fbTrendLogger(
    VI_System_Time_MS := GVL_TIME_SERVICE.G_Now_MS,
    VI_Config := L_TrendConfig,
    VI_Current_Value := GVL_STATE.G_Room_Temps[1],
    VO_Data => L_TrendData
);

fbTrendAdapter(
    VI_Data := L_TrendData,
    VO_Average => L_Average,
    VO_Min => L_Min,
    VO_Max => L_Max,
    VO_Trend_Up => L_Trend_Up,
    VO_Trend_Down => L_Trend_Down
);
          
END_PROGRAM

PROGRAM PRG_Peer_Session_Publication

            // ======================================================
// PEER SESSION PUBLICATION
// ======================================================
// Canonical local PLC session export.
//
// Purpose:
// publish normalized runtime/session authority state into
// explicit peer-session transport contract surface.
//
// This layer does NOT:
// - perform network replication
// - perform distributed reconciliation
// - consume remote peer state
//
// Future transport/replication layers may replicate these
// fields to partner PLCs or external HA channels.
// ======================================================

GVL_PEER_SESSION.Remote_Session_Valid :=
    GVL_RUNTIME_EPOCH.Runtime_Runtime_Barrier_OK
    AND GVL_RUNTIME_EPOCH.Runtime_IO_Publication_Allowed;

GVL_PEER_SESSION.Remote_Last_Refresh_MS :=
    GVL_STATUS.G_System_Time_MS;

GVL_PEER_SESSION.Remote_Runtime_Epoch :=
    GVL_RUNTIME_EPOCH.Runtime_Epoch;

GVL_PEER_SESSION.Remote_Snapshot_Epoch :=
    GVL_RUNTIME_SNAPSHOT.Snapshot_Epoch;

GVL_PEER_SESSION.Remote_Boot_Generation :=
    GVL_TIME_MONOTONIC.Boot_Generation_ID;

GVL_PEER_SESSION.Remote_Fencing_Token :=
    GVL_PLC_FENCING.PLC_Fencing_Token;

GVL_PEER_SESSION.Remote_Publication_Allowed :=
    GVL_OUTPUT_EPOCH.Output_Publication_Valid
    AND NOT GVL_OUTPUT_EPOCH.Output_Forced_Safe_Decay;

GVL_PEER_SESSION.Remote_Runtime_Healthy :=
    GVL_RUNTIME_EPOCH.Runtime_Runtime_Barrier_OK;

// >>> BULK_SYNC_ANCHOR: PRG_Peer_Session_Publication <<<
          
END_PROGRAM

PROGRAM PRG_PLC_Arbitration

            // Update heartbeat
IF GVL_STATUS.G_Remote_PLC_Pulse THEN
    GVL_STATUS.G_Remote_PLC_Last_Seen_MS := GVL_TIME_SERVICE.G_Now_MS;
END_IF;

// Alive check (3s)
GVL_STATUS.G_Remote_PLC_Alive :=
    (GVL_TIME_SERVICE.G_Now_MS - GVL_STATUS.G_Remote_PLC_Last_Seen_MS) < 3000;

// Deterministic arbitration.
// If remote is not alive, local PLC owns runtime.
// If remote is alive, the lowest PLC ID wins; equality keeps local active
// because G_Active_PLC_ID defaults to the configured local owner ID.
IF NOT GVL_STATUS.G_Remote_PLC_Alive THEN
    GVL_STATUS.G_Is_Active_PLC := TRUE;
    GVL_STATUS.G_Active_PLC_ID := GVL_STATUS.G_Local_PLC_ID;
ELSE
    IF GVL_STATUS.G_Local_PLC_ID <= GVL_STATUS.G_Active_PLC_ID THEN
        GVL_STATUS.G_Is_Active_PLC := TRUE;
        GVL_STATUS.G_Active_PLC_ID := GVL_STATUS.G_Local_PLC_ID;
    ELSE
        GVL_STATUS.G_Is_Active_PLC := FALSE;
    END_IF;
END_IF;

GVL_STATUS.G_Other_PLC_Is_Active :=
    GVL_STATUS.G_Remote_PLC_Alive AND NOT GVL_STATUS.G_Is_Active_PLC;

// >>> BULK_SYNC_ANCHOR: PRG_PLC_Arbitration <<<
          
END_PROGRAM

PROGRAM PRG_Physical_Snapshot_Governor
  VAR
    L_Now_MS : UDINT;
    L_Snapshot_Valid : BOOL := TRUE;
    L_Error_Code : UDINT := 0;
    L_Error_Text : STRING(160) := '';
  END_VAR

            L_Now_MS := GVL_STATUS.G_System_Time_MS;
L_Snapshot_Valid := TRUE;
L_Error_Code := 0;
L_Error_Text := '';

GVL_PHYSICAL_SNAPSHOT.Physical_Snapshot_Valid := FALSE;
GVL_PHYSICAL_SNAPSHOT.Physical_Snapshot_Frozen := FALSE;
GVL_PHYSICAL_SNAPSHOT.Physical_Snapshot_Publication_Allowed := FALSE;
GVL_PHYSICAL_SNAPSHOT.Physical_Snapshot_Isolation_Valid := FALSE;
GVL_PHYSICAL_SNAPSHOT.Physical_Snapshot_Copy_Valid := FALSE;
GVL_PHYSICAL_SNAPSHOT.Physical_Snapshot_Freshness_Valid := FALSE;
GVL_PHYSICAL_SNAPSHOT.Physical_Snapshot_Consensus_Coherent := FALSE;
GVL_PHYSICAL_SNAPSHOT.Physical_Snapshot_Causality_Coherent := FALSE;

GVL_PHYSICAL_SNAPSHOT.Physical_Snapshot_Runtime_Epoch := ULINT_TO_UDINT(GVL_RUNTIME_EPOCH.Runtime_Epoch);
GVL_PHYSICAL_SNAPSHOT.Physical_Snapshot_Output_Epoch := ULINT_TO_UDINT(GVL_OUTPUT_EPOCH.Output_Publication_Epoch);

IF NOT GVL_RUNTIME_EPOCH.Runtime_Runtime_Barrier_OK THEN
    L_Snapshot_Valid := FALSE;
    L_Error_Code := 23000;
    L_Error_Text := 'Physical snapshot runtime barrier invalid';
END_IF;

IF L_Snapshot_Valid AND NOT GVL_OUTPUT_EPOCH.Output_Publication_Valid THEN
    L_Snapshot_Valid := FALSE;
    L_Error_Code := 23001;
    L_Error_Text := 'Physical snapshot output publication invalid';
END_IF;

IF L_Snapshot_Valid AND GVL_PHYSICAL_SNAPSHOT.Physical_Snapshot_Mutation_Detected THEN
    L_Snapshot_Valid := FALSE;
    L_Error_Code := 23002;
    L_Error_Text := 'Physical snapshot mutation detected';
END_IF;

IF L_Snapshot_Valid AND GVL_PHYSICAL_SNAPSHOT.Physical_Snapshot_Replay_Suspected THEN
    L_Snapshot_Valid := FALSE;
    L_Error_Code := 23003;
    L_Error_Text := 'Physical snapshot replay suspected';
END_IF;

IF L_Snapshot_Valid AND GVL_PHYSICAL_SNAPSHOT.Physical_Snapshot_Lease_Expired THEN
    L_Snapshot_Valid := FALSE;
    L_Error_Code := 23004;
    L_Error_Text := 'Physical snapshot lease expired';
END_IF;

IF L_Snapshot_Valid THEN
    GVL_PHYSICAL_SNAPSHOT.Physical_Snapshot_Valid := TRUE;
    GVL_PHYSICAL_SNAPSHOT.Physical_Snapshot_Frozen := TRUE;
    GVL_PHYSICAL_SNAPSHOT.Physical_Snapshot_Publication_Allowed := TRUE;
    GVL_PHYSICAL_SNAPSHOT.Physical_Snapshot_Isolation_Valid := TRUE;
    GVL_PHYSICAL_SNAPSHOT.Physical_Snapshot_Copy_Valid := TRUE;
    GVL_PHYSICAL_SNAPSHOT.Physical_Snapshot_Freshness_Valid := TRUE;
    GVL_PHYSICAL_SNAPSHOT.Physical_Snapshot_Consensus_Coherent := TRUE;
    GVL_PHYSICAL_SNAPSHOT.Physical_Snapshot_Causality_Coherent := TRUE;
    GVL_PHYSICAL_SNAPSHOT.Physical_Snapshot_Epoch := GVL_PHYSICAL_SNAPSHOT.Physical_Snapshot_Epoch + 1;
    GVL_PHYSICAL_SNAPSHOT.Physical_Snapshot_Last_Update_MS := L_Now_MS;
    GVL_PHYSICAL_SNAPSHOT.Physical_Snapshot_Last_Error_Code := 0;
    GVL_PHYSICAL_SNAPSHOT.Physical_Snapshot_Last_Error_Text := '';
ELSE
    GVL_PHYSICAL_SNAPSHOT.Physical_Snapshot_Valid := FALSE;
    GVL_PHYSICAL_SNAPSHOT.Physical_Snapshot_Frozen := FALSE;
    GVL_PHYSICAL_SNAPSHOT.Physical_Snapshot_Publication_Allowed := FALSE;
    GVL_PHYSICAL_SNAPSHOT.Physical_Snapshot_Last_Error_Code := L_Error_Code;
    GVL_PHYSICAL_SNAPSHOT.Physical_Snapshot_Last_Error_Text := L_Error_Text;
    GVL_PHYSICAL_SNAPSHOT.Physical_Snapshot_Invalidation_Count := GVL_PHYSICAL_SNAPSHOT.Physical_Snapshot_Invalidation_Count + 1;
END_IF;
          
END_PROGRAM

PROGRAM PRG_Causality_Reversal_Prevention_Governor

            IF GVL_HISTORICAL_ORDERING_INTEGRITY_FABRIC.Historical_Ordering_Integrity_Granted
AND NOT GVL_CAUSALITY_REVERSAL_PREVENTION_FABRIC.Causality_Reversal_Detected
AND NOT GVL_CAUSALITY_REVERSAL_PREVENTION_FABRIC.Resurrection_After_Revocation_Detected
AND NOT GVL_CAUSALITY_REVERSAL_PREVENTION_FABRIC.Unsafe_Temporal_Replay_Detected THEN

    GVL_CAUSALITY_REVERSAL_PREVENTION_FABRIC.Causality_Reversal_Prevention_Valid := TRUE;
    GVL_CAUSALITY_REVERSAL_PREVENTION_FABRIC.Causality_Reversal_Prevention_Granted := TRUE;
    GVL_CAUSALITY_REVERSAL_PREVENTION_FABRIC.Causality_Reversal_Prevented := TRUE;
    GVL_CAUSALITY_REVERSAL_PREVENTION_FABRIC.Authority_Ordering_Canonical := TRUE;
    GVL_CAUSALITY_REVERSAL_PREVENTION_FABRIC.Revocation_Resurrection_Boundary_Stable := TRUE;
END_IF;
          
END_PROGRAM

PROGRAM PRG_Epistemic_Integrity_Governor
  VAR
    L_Now_MS : UDINT;
    L_Epistemic_Valid : BOOL := TRUE;
    L_Error_Code : UDINT := 0;
    L_Error_Text : STRING(160) := '';
  END_VAR

            L_Now_MS := GVL_STATUS.G_System_Time_MS;
L_Epistemic_Valid := TRUE;
L_Error_Code := 0;
L_Error_Text := '';

// Fail-safe defaults.
GVL_EPISTEMIC_INTEGRITY_FABRIC.Epistemic_Integrity_Valid := FALSE;
GVL_EPISTEMIC_INTEGRITY_FABRIC.Epistemic_Integrity_Granted := FALSE;
GVL_EPISTEMIC_INTEGRITY_FABRIC.Epistemic_Integrity_Quarantine_Active := TRUE;

GVL_EPISTEMIC_INTEGRITY_FABRIC.Physical_Reality_Model_Coherent := FALSE;
GVL_EPISTEMIC_INTEGRITY_FABRIC.Sensor_Truth_Consensus_Valid := FALSE;
GVL_EPISTEMIC_INTEGRITY_FABRIC.Telemetry_Reality_Alignment_Stable := FALSE;
GVL_EPISTEMIC_INTEGRITY_FABRIC.Distributed_Reality_Model_Consistent := FALSE;
GVL_EPISTEMIC_INTEGRITY_FABRIC.Causal_Model_Physically_Valid := FALSE;

// Forensic evidence required.
IF NOT GVL_FORENSIC_EVIDENCE_FABRIC.Forensic_Evidence_Granted THEN
    L_Epistemic_Valid := FALSE;
    L_Error_Code := 44000;
    L_Error_Text := 'Forensic evidence authority not granted';
END_IF;

// Epistemic split-brain detectors.
IF GVL_EPISTEMIC_INTEGRITY_FABRIC.Physically_False_Consensus_Detected THEN
    L_Epistemic_Valid := FALSE;
    L_Error_Code := 44001;
    L_Error_Text := 'Physically false consensus detected';
END_IF;

IF GVL_EPISTEMIC_INTEGRITY_FABRIC.Telemetry_Corruption_Coherent_Detected THEN
    L_Epistemic_Valid := FALSE;
    L_Error_Code := 44002;
    L_Error_Text := 'Telemetry corruption coherence detected';
END_IF;

IF GVL_EPISTEMIC_INTEGRITY_FABRIC.Historical_Reality_Divergence_Detected THEN
    L_Epistemic_Valid := FALSE;
    L_Error_Code := 44003;
    L_Error_Text := 'Historical reality divergence detected';
END_IF;

IF GVL_EPISTEMIC_INTEGRITY_FABRIC.Sensor_Trust_Erosion_Detected THEN
    L_Epistemic_Valid := FALSE;
    L_Error_Code := 44004;
    L_Error_Text := 'Sensor trust erosion detected';
END_IF;

IF GVL_EPISTEMIC_INTEGRITY_FABRIC.Causal_Model_Poisoning_Detected THEN
    L_Epistemic_Valid := FALSE;
    L_Error_Code := 44005;
    L_Error_Text := 'Causal model poisoning detected';
END_IF;

IF GVL_EPISTEMIC_INTEGRITY_FABRIC.LongTerm_Epistemic_Drift_Detected THEN
    L_Epistemic_Valid := FALSE;
    L_Error_Code := 44006;
    L_Error_Text := 'Long-term epistemic drift detected';
END_IF;

// Physical reality anchoring validation.
IF L_Epistemic_Valid
AND NOT GVL_EPISTEMIC_INTEGRITY_FABRIC.Historical_Reality_Anchoring_Valid THEN
    L_Epistemic_Valid := FALSE;
    L_Error_Code := 44010;
    L_Error_Text := 'Historical reality anchoring invalid';
END_IF;

IF L_Epistemic_Valid
AND NOT GVL_EPISTEMIC_INTEGRITY_FABRIC.Physical_Truth_Lineage_Coherent THEN
    L_Epistemic_Valid := FALSE;
    L_Error_Code := 44011;
    L_Error_Text := 'Physical truth lineage coherence invalid';
END_IF;

IF L_Epistemic_Valid
AND NOT GVL_EPISTEMIC_INTEGRITY_FABRIC.Reality_Model_Drift_Bounded THEN
    L_Epistemic_Valid := FALSE;
    L_Error_Code := 44012;
    L_Error_Text := 'Reality model drift bounds invalid';
END_IF;

IF L_Epistemic_Valid
AND NOT GVL_EPISTEMIC_INTEGRITY_FABRIC.Semantic_To_Physical_Causality_Valid THEN
    L_Epistemic_Valid := FALSE;
    L_Error_Code := 44013;
    L_Error_Text := 'Semantic-to-physical causality invalid';
END_IF;

IF L_Epistemic_Valid THEN
    GVL_EPISTEMIC_INTEGRITY_FABRIC.Epistemic_Integrity_Valid := TRUE;
    GVL_EPISTEMIC_INTEGRITY_FABRIC.Epistemic_Integrity_Granted := TRUE;
    GVL_EPISTEMIC_INTEGRITY_FABRIC.Epistemic_Integrity_Quarantine_Active := FALSE;

    GVL_EPISTEMIC_INTEGRITY_FABRIC.Physical_Reality_Model_Coherent := TRUE;
    GVL_EPISTEMIC_INTEGRITY_FABRIC.Sensor_Truth_Consensus_Valid := TRUE;
    GVL_EPISTEMIC_INTEGRITY_FABRIC.Telemetry_Reality_Alignment_Stable := TRUE;
    GVL_EPISTEMIC_INTEGRITY_FABRIC.Distributed_Reality_Model_Consistent := TRUE;
    GVL_EPISTEMIC_INTEGRITY_FABRIC.Causal_Model_Physically_Valid := TRUE;

    GVL_EPISTEMIC_INTEGRITY_FABRIC.Epistemic_Integrity_Epoch :=
        GVL_FORENSIC_EVIDENCE_FABRIC.Forensic_Evidence_Epoch;

    GVL_EPISTEMIC_INTEGRITY_FABRIC.Epistemic_Integrity_Epoch_Coherent := TRUE;

    GVL_EPISTEMIC_INTEGRITY_FABRIC.Epistemic_Integrity_Last_Update_MS :=
        L_Now_MS;

    GVL_EPISTEMIC_INTEGRITY_FABRIC.Epistemic_Integrity_Lease_Expired := FALSE;

    GVL_EPISTEMIC_INTEGRITY_FABRIC.Epistemic_Integrity_Last_Error_Code := 0;
    GVL_EPISTEMIC_INTEGRITY_FABRIC.Epistemic_Integrity_Last_Error_Text := '';
ELSE
    GVL_EPISTEMIC_INTEGRITY_FABRIC.Epistemic_Integrity_Valid := FALSE;
    GVL_EPISTEMIC_INTEGRITY_FABRIC.Epistemic_Integrity_Granted := FALSE;
    GVL_EPISTEMIC_INTEGRITY_FABRIC.Epistemic_Integrity_Quarantine_Active := TRUE;

    GVL_EPISTEMIC_INTEGRITY_FABRIC.Epistemic_Integrity_Lease_Expired := TRUE;

    GVL_EPISTEMIC_INTEGRITY_FABRIC.Epistemic_Integrity_Last_Error_Code :=
        L_Error_Code;

    GVL_EPISTEMIC_INTEGRITY_FABRIC.Epistemic_Integrity_Last_Error_Text :=
        L_Error_Text;

    GVL_EPISTEMIC_INTEGRITY_FABRIC.Epistemic_Integrity_Invalidation_Count :=
        GVL_EPISTEMIC_INTEGRITY_FABRIC.Epistemic_Integrity_Invalidation_Count + 1;
END_IF;
          
END_PROGRAM

PROGRAM PRG_Authority_Provenance_Governor
  VAR
    L_Now_MS : UDINT;
    L_Provenance_Valid : BOOL := TRUE;
    L_Error_Code : UDINT := 0;
    L_Error_Text : STRING(160) := '';
  END_VAR

            L_Now_MS := GVL_STATUS.G_System_Time_MS;
L_Provenance_Valid := TRUE;
L_Error_Code := 0;
L_Error_Text := '';

// Fail-safe defaults.
GVL_AUTHORITY_PROVENANCE_FABRIC.Authority_Provenance_Valid := FALSE;
GVL_AUTHORITY_PROVENANCE_FABRIC.Authority_Provenance_Granted := FALSE;
GVL_AUTHORITY_PROVENANCE_FABRIC.Authority_Provenance_Quarantine_Active := TRUE;

GVL_AUTHORITY_PROVENANCE_FABRIC.Bootstrap_Authority_Authentic := FALSE;
GVL_AUTHORITY_PROVENANCE_FABRIC.Commissioning_Lineage_Traceable := FALSE;
GVL_AUTHORITY_PROVENANCE_FABRIC.Trust_Seed_Integrity_Valid := FALSE;
GVL_AUTHORITY_PROVENANCE_FABRIC.Root_Authority_Attribution_Coherent := FALSE;
GVL_AUTHORITY_PROVENANCE_FABRIC.Provenance_Causality_Grounded := FALSE;

// Meta-governance required.
IF NOT GVL_META_GOVERNANCE_FABRIC.Meta_Governance_Granted THEN
    L_Provenance_Valid := FALSE;
    L_Error_Code := 46000;
    L_Error_Text := 'Meta-governance authority not granted';
END_IF;

// Authority-origin split-brain detectors.
IF GVL_AUTHORITY_PROVENANCE_FABRIC.Bootstrap_Identity_Corruption_Detected THEN
    L_Provenance_Valid := FALSE;
    L_Error_Code := 46001;
    L_Error_Text := 'Bootstrap identity corruption detected';
END_IF;

IF GVL_AUTHORITY_PROVENANCE_FABRIC.Forged_Authority_Root_Detected THEN
    L_Provenance_Valid := FALSE;
    L_Error_Code := 46002;
    L_Error_Text := 'Forged authority root detected';
END_IF;

IF GVL_AUTHORITY_PROVENANCE_FABRIC.Commissioning_Provenance_Gap_Detected THEN
    L_Provenance_Valid := FALSE;
    L_Error_Code := 46003;
    L_Error_Text := 'Commissioning provenance gap detected';
END_IF;

IF GVL_AUTHORITY_PROVENANCE_FABRIC.Trust_Seed_Impersonation_Detected THEN
    L_Provenance_Valid := FALSE;
    L_Error_Code := 46004;
    L_Error_Text := 'Trust seed impersonation detected';
END_IF;

IF GVL_AUTHORITY_PROVENANCE_FABRIC.Origin_Authenticity_Erosion_Detected THEN
    L_Provenance_Valid := FALSE;
    L_Error_Code := 46005;
    L_Error_Text := 'Origin authenticity erosion detected';
END_IF;

IF GVL_AUTHORITY_PROVENANCE_FABRIC.Root_Lineage_Tampering_Detected THEN
    L_Provenance_Valid := FALSE;
    L_Error_Code := 46006;
    L_Error_Text := 'Root lineage tampering detected';
END_IF;

// Provenance integrity validation.
IF L_Provenance_Valid
AND NOT GVL_AUTHORITY_PROVENANCE_FABRIC.Historical_Origin_Lineage_Valid THEN
    L_Provenance_Valid := FALSE;
    L_Error_Code := 46010;
    L_Error_Text := 'Historical origin lineage invalid';
END_IF;

IF L_Provenance_Valid
AND NOT GVL_AUTHORITY_PROVENANCE_FABRIC.Distributed_Trust_Chain_Coherent THEN
    L_Provenance_Valid := FALSE;
    L_Error_Code := 46011;
    L_Error_Text := 'Distributed trust chain coherence invalid';
END_IF;

IF L_Provenance_Valid
AND NOT GVL_AUTHORITY_PROVENANCE_FABRIC.Authority_Origin_Continuity_Stable THEN
    L_Provenance_Valid := FALSE;
    L_Error_Code := 46012;
    L_Error_Text := 'Authority origin continuity invalid';
END_IF;

IF L_Provenance_Valid
AND NOT GVL_AUTHORITY_PROVENANCE_FABRIC.Root_Identity_Cryptographic_Validity THEN
    L_Provenance_Valid := FALSE;
    L_Error_Code := 46013;
    L_Error_Text := 'Root identity cryptographic validity invalid';
END_IF;

IF L_Provenance_Valid THEN
    GVL_AUTHORITY_PROVENANCE_FABRIC.Authority_Provenance_Valid := TRUE;
    GVL_AUTHORITY_PROVENANCE_FABRIC.Authority_Provenance_Granted := TRUE;
    GVL_AUTHORITY_PROVENANCE_FABRIC.Authority_Provenance_Quarantine_Active := FALSE;

    GVL_AUTHORITY_PROVENANCE_FABRIC.Bootstrap_Authority_Authentic := TRUE;
    GVL_AUTHORITY_PROVENANCE_FABRIC.Commissioning_Lineage_Traceable := TRUE;
    GVL_AUTHORITY_PROVENANCE_FABRIC.Trust_Seed_Integrity_Valid := TRUE;
    GVL_AUTHORITY_PROVENANCE_FABRIC.Root_Authority_Attribution_Coherent := TRUE;
    GVL_AUTHORITY_PROVENANCE_FABRIC.Provenance_Causality_Grounded := TRUE;

    GVL_AUTHORITY_PROVENANCE_FABRIC.Authority_Provenance_Epoch :=
        GVL_META_GOVERNANCE_FABRIC.Meta_Governance_Epoch;

    GVL_AUTHORITY_PROVENANCE_FABRIC.Authority_Provenance_Epoch_Coherent := TRUE;

    GVL_AUTHORITY_PROVENANCE_FABRIC.Authority_Provenance_Last_Update_MS :=
        L_Now_MS;

    GVL_AUTHORITY_PROVENANCE_FABRIC.Authority_Provenance_Lease_Expired := FALSE;

    GVL_AUTHORITY_PROVENANCE_FABRIC.Authority_Provenance_Last_Error_Code := 0;
    GVL_AUTHORITY_PROVENANCE_FABRIC.Authority_Provenance_Last_Error_Text := '';
ELSE
    GVL_AUTHORITY_PROVENANCE_FABRIC.Authority_Provenance_Valid := FALSE;
    GVL_AUTHORITY_PROVENANCE_FABRIC.Authority_Provenance_Granted := FALSE;
    GVL_AUTHORITY_PROVENANCE_FABRIC.Authority_Provenance_Quarantine_Active := TRUE;

    GVL_AUTHORITY_PROVENANCE_FABRIC.Authority_Provenance_Lease_Expired := TRUE;

    GVL_AUTHORITY_PROVENANCE_FABRIC.Authority_Provenance_Last_Error_Code :=
        L_Error_Code;

    GVL_AUTHORITY_PROVENANCE_FABRIC.Authority_Provenance_Last_Error_Text :=
        L_Error_Text;

    GVL_AUTHORITY_PROVENANCE_FABRIC.Authority_Provenance_Invalidation_Count :=
        GVL_AUTHORITY_PROVENANCE_FABRIC.Authority_Provenance_Invalidation_Count + 1;
END_IF;
          
END_PROGRAM

PROGRAM PRG_System_Evacuation
  VAR
    fbSystemEvacuation : FB_System_Evacuation;
  END_VAR

            fbSystemEvacuation();
          
END_PROGRAM

PROGRAM PRG_Peer_Heartbeat_Ingestion
  VAR
    L_Now_MS : UDINT;
  END_VAR

            // ======================================================
// PEER HEARTBEAT INGESTION
// ======================================================
// Bounded transport/heartbeat ingestion bridge.
//
// Purpose:
// map physical partner heartbeat inputs into runtime-visible
// remote PLC liveness state consumed by arbitration layers.
//
// This layer does NOT:
// - perform distributed epoch reconciliation
// - publish peer fencing tokens
// - mutate distributed authority state
// - participate in runtime/output hard-stop governance
//
// Ownership:
// physical partner inputs  -> GVL_IO
// heartbeat ingestion      -> this PRG
// arbitration/governance   -> downstream consumers only
// ======================================================

L_Now_MS := GVL_STATUS.G_System_Time_MS;

// ------------------------------------------------------
// Physical heartbeat ingestion.
// ------------------------------------------------------

GVL_STATUS.G_Remote_PLC_Pulse := GVL_IO.DI_Partner_Pulse;

// ------------------------------------------------------
// Partner active visibility projection.
// ------------------------------------------------------

IF GVL_IO.DI_Partner_Active THEN
    GVL_STATUS.G_Remote_PLC_Last_Seen_MS := L_Now_MS;
END_IF;

// ------------------------------------------------------
// Optional pulse freshness refresh.
// ------------------------------------------------------

IF GVL_IO.DI_Partner_Pulse THEN
    GVL_STATUS.G_Remote_PLC_Last_Seen_MS := L_Now_MS;
END_IF;

// ------------------------------------------------------
// Remote liveness projection.
// ------------------------------------------------------

GVL_STATUS.G_Remote_PLC_Alive :=
    (L_Now_MS - GVL_STATUS.G_Remote_PLC_Last_Seen_MS) < 3000;

// >>> BULK_SYNC_ANCHOR: PRG_Peer_Heartbeat_Ingestion <<<
          
END_PROGRAM

PROGRAM PRG_Compliance_Federation_Governor
  VAR
    L_Now_MS : UDINT;
    L_Compliance_Valid : BOOL := TRUE;
    L_Error_Code : UDINT := 0;
    L_Error_Text : STRING(160) := '';
  END_VAR

            L_Now_MS := GVL_STATUS.G_System_Time_MS;
L_Compliance_Valid := TRUE;
L_Error_Code := 0;
L_Error_Text := '';

// Fail-safe defaults.
GVL_COMPLIANCE_FEDERATION_FABRIC.Compliance_Federation_Valid := FALSE;
GVL_COMPLIANCE_FEDERATION_FABRIC.Compliance_Federation_Granted := FALSE;
GVL_COMPLIANCE_FEDERATION_FABRIC.Compliance_Federation_Quarantine_Active := TRUE;

GVL_COMPLIANCE_FEDERATION_FABRIC.Regulatory_Semantics_Coherent := FALSE;
GVL_COMPLIANCE_FEDERATION_FABRIC.Certification_Boundary_Valid := FALSE;
GVL_COMPLIANCE_FEDERATION_FABRIC.Regional_Safety_Envelope_Aligned := FALSE;
GVL_COMPLIANCE_FEDERATION_FABRIC.Governance_Trust_Boundary_Stable := FALSE;
GVL_COMPLIANCE_FEDERATION_FABRIC.Policy_Compliance_Coherent := FALSE;

// Semantic federation required.
IF NOT GVL_SEMANTIC_FEDERATION_FABRIC.Semantic_Federation_Granted THEN
    L_Compliance_Valid := FALSE;
    L_Error_Code := 42000;
    L_Error_Text := 'Semantic federation authority not granted';
END_IF;

// Regulatory semantic split-brain detectors.
IF GVL_COMPLIANCE_FEDERATION_FABRIC.CrossJurisdiction_Semantic_Drift_Detected THEN
    L_Compliance_Valid := FALSE;
    L_Error_Code := 42001;
    L_Error_Text := 'Cross-jurisdiction semantic drift detected';
END_IF;

IF GVL_COMPLIANCE_FEDERATION_FABRIC.Certification_Boundary_Violation_Detected THEN
    L_Compliance_Valid := FALSE;
    L_Error_Code := 42002;
    L_Error_Text := 'Certification boundary violation detected';
END_IF;

IF GVL_COMPLIANCE_FEDERATION_FABRIC.Policy_Compliance_Divergence_Detected THEN
    L_Compliance_Valid := FALSE;
    L_Error_Code := 42003;
    L_Error_Text := 'Policy compliance divergence detected';
END_IF;

IF GVL_COMPLIANCE_FEDERATION_FABRIC.Regional_Safety_Envelope_Mismatch_Detected THEN
    L_Compliance_Valid := FALSE;
    L_Error_Code := 42004;
    L_Error_Text := 'Regional safety envelope mismatch detected';
END_IF;

IF GVL_COMPLIANCE_FEDERATION_FABRIC.Regulatory_Trust_Corruption_Detected THEN
    L_Compliance_Valid := FALSE;
    L_Error_Code := 42005;
    L_Error_Text := 'Regulatory trust corruption detected';
END_IF;

IF GVL_COMPLIANCE_FEDERATION_FABRIC.Governance_Authority_Leakage_Detected THEN
    L_Compliance_Valid := FALSE;
    L_Error_Code := 42006;
    L_Error_Text := 'Governance authority leakage detected';
END_IF;

// Compliance federation validation.
IF L_Compliance_Valid
AND NOT GVL_COMPLIANCE_FEDERATION_FABRIC.CrossJurisdiction_Authority_Aligned THEN
    L_Compliance_Valid := FALSE;
    L_Error_Code := 42010;
    L_Error_Text := 'Cross-jurisdiction authority alignment invalid';
END_IF;

IF L_Compliance_Valid
AND NOT GVL_COMPLIANCE_FEDERATION_FABRIC.Compliance_Runtime_Projection_Stable THEN
    L_Compliance_Valid := FALSE;
    L_Error_Code := 42011;
    L_Error_Text := 'Compliance runtime projection unstable';
END_IF;

IF L_Compliance_Valid
AND NOT GVL_COMPLIANCE_FEDERATION_FABRIC.External_Governance_Interpretation_Valid THEN
    L_Compliance_Valid := FALSE;
    L_Error_Code := 42012;
    L_Error_Text := 'External governance interpretation invalid';
END_IF;

IF L_Compliance_Valid
AND NOT GVL_COMPLIANCE_FEDERATION_FABRIC.Certified_Operational_Semantics_Valid THEN
    L_Compliance_Valid := FALSE;
    L_Error_Code := 42013;
    L_Error_Text := 'Certified operational semantics invalid';
END_IF;

IF L_Compliance_Valid THEN
    GVL_COMPLIANCE_FEDERATION_FABRIC.Compliance_Federation_Valid := TRUE;
    GVL_COMPLIANCE_FEDERATION_FABRIC.Compliance_Federation_Granted := TRUE;
    GVL_COMPLIANCE_FEDERATION_FABRIC.Compliance_Federation_Quarantine_Active := FALSE;

    GVL_COMPLIANCE_FEDERATION_FABRIC.Regulatory_Semantics_Coherent := TRUE;
    GVL_COMPLIANCE_FEDERATION_FABRIC.Certification_Boundary_Valid := TRUE;
    GVL_COMPLIANCE_FEDERATION_FABRIC.Regional_Safety_Envelope_Aligned := TRUE;
    GVL_COMPLIANCE_FEDERATION_FABRIC.Governance_Trust_Boundary_Stable := TRUE;
    GVL_COMPLIANCE_FEDERATION_FABRIC.Policy_Compliance_Coherent := TRUE;

    GVL_COMPLIANCE_FEDERATION_FABRIC.Compliance_Federation_Epoch :=
        GVL_SEMANTIC_FEDERATION_FABRIC.Semantic_Federation_Epoch;

    GVL_COMPLIANCE_FEDERATION_FABRIC.Compliance_Federation_Epoch_Coherent := TRUE;

    GVL_COMPLIANCE_FEDERATION_FABRIC.Compliance_Federation_Last_Update_MS :=
        L_Now_MS;

    GVL_COMPLIANCE_FEDERATION_FABRIC.Compliance_Federation_Lease_Expired := FALSE;

    GVL_COMPLIANCE_FEDERATION_FABRIC.Compliance_Federation_Last_Error_Code := 0;
    GVL_COMPLIANCE_FEDERATION_FABRIC.Compliance_Federation_Last_Error_Text := '';
ELSE
    GVL_COMPLIANCE_FEDERATION_FABRIC.Compliance_Federation_Valid := FALSE;
    GVL_COMPLIANCE_FEDERATION_FABRIC.Compliance_Federation_Granted := FALSE;
    GVL_COMPLIANCE_FEDERATION_FABRIC.Compliance_Federation_Quarantine_Active := TRUE;

    GVL_COMPLIANCE_FEDERATION_FABRIC.Compliance_Federation_Lease_Expired := TRUE;

    GVL_COMPLIANCE_FEDERATION_FABRIC.Compliance_Federation_Last_Error_Code :=
        L_Error_Code;

    GVL_COMPLIANCE_FEDERATION_FABRIC.Compliance_Federation_Last_Error_Text :=
        L_Error_Text;

    GVL_COMPLIANCE_FEDERATION_FABRIC.Compliance_Federation_Invalidation_Count :=
        GVL_COMPLIANCE_FEDERATION_FABRIC.Compliance_Federation_Invalidation_Count + 1;
END_IF;
          
END_PROGRAM

PROGRAM PRG_Distributed_Forward_Progress_Governor

            IF GVL_RESOURCE_STARVATION_BOUNDARY_FABRIC.Resource_Starvation_Boundary_Granted
AND NOT GVL_DISTRIBUTED_FORWARD_PROGRESS_FABRIC.Distributed_Livelock_Detected
AND NOT GVL_DISTRIBUTED_FORWARD_PROGRESS_FABRIC.Cluster_Progress_Fork_Detected
AND NOT GVL_DISTRIBUTED_FORWARD_PROGRESS_FABRIC.Distributed_Consensus_Progress_Deadlock THEN

    GVL_DISTRIBUTED_FORWARD_PROGRESS_FABRIC.Distributed_Forward_Progress_Valid := TRUE;
    GVL_DISTRIBUTED_FORWARD_PROGRESS_FABRIC.Distributed_Forward_Progress_Granted := TRUE;
    GVL_DISTRIBUTED_FORWARD_PROGRESS_FABRIC.Distributed_Forward_Progress_Canonical := TRUE;
    GVL_DISTRIBUTED_FORWARD_PROGRESS_FABRIC.Cluster_Progress_Consensus_Stable := TRUE;
    GVL_DISTRIBUTED_FORWARD_PROGRESS_FABRIC.Distributed_Recovery_Progress_Valid := TRUE;
END_IF;
          
END_PROGRAM

PROGRAM PRG_Recovery_Cleanup_Governor
  VAR
    L_Now_MS : UDINT;
    L_Recovery_Valid : BOOL := TRUE;
    L_Error_Code : UDINT := 0;
    L_Error_Text : STRING(160) := '';
    L_Distributed_Recovery_Allowed : BOOL;
    L_Cluster_Recovery_Lock : BOOL;
    L_Cluster_Quarantine : BOOL;
    L_Finalized_Publication_Continuity : BOOL;
  END_VAR

            L_Now_MS := GVL_STATUS.G_System_Time_MS;
L_Recovery_Valid := TRUE;
L_Error_Code := 0;
L_Error_Text := '';

GVL_RECOVERY_GOVERNANCE.Recovery_Semantic_Residue_Detected := FALSE;
GVL_RECOVERY_GOVERNANCE.Recovery_Degraded_State_Residual := FALSE;
GVL_RECOVERY_GOVERNANCE.Recovery_Retained_State_Residual := FALSE;

L_Distributed_Recovery_Allowed :=
    GVL_Distributed_Execution_Gates.G_Can_Recover;

L_Cluster_Recovery_Lock :=
    GVL_Cluster_Runtime_FSM.G_State_Recovery_Lock;

L_Cluster_Quarantine :=
    GVL_Cluster_Runtime_FSM.G_State_Quarantine;

// Finalized publication continuity.
L_Finalized_Publication_Continuity :=
    GVL_DISTRIBUTED_SNAPSHOT.Distributed_Publication_Reconciled
    AND GVL_DISTRIBUTED_SNAPSHOT.Distributed_Publication_Freeze_Valid
    AND GVL_DISTRIBUTED_SNAPSHOT.Distributed_Snapshot_Consistent
    AND GVL_DISTRIBUTED_COMMIT.Distributed_Commit_Valid
    AND NOT GVL_DISTRIBUTED_COMMIT.Commit_Lease_Expired
    AND GVL_OUTPUT_EPOCH.Output_Publication_Valid
    AND GVL_OUTPUT_EPOCH.Output_Runtime_Epoch_Valid
    AND NOT GVL_OUTPUT_EPOCH.Output_Lease_Expired
    AND NOT GVL_OUTPUT_EPOCH.Output_Forced_Safe_Decay;

IF NOT GVL_TIME_MONOTONIC.Monotonic_Time_Valid THEN
    L_Recovery_Valid := FALSE;
    L_Error_Code := 9001;
    L_Error_Text := 'Recovery monotonic authority invalid';
END_IF;

IF L_Recovery_Valid
   AND NOT L_Distributed_Recovery_Allowed THEN

    L_Recovery_Valid := FALSE;

    L_Error_Code := 9010;
    L_Error_Text :=
        'Distributed recovery governance restricted';

END_IF;

IF L_Recovery_Valid
   AND L_Cluster_Recovery_Lock THEN

    L_Recovery_Valid := FALSE;

    L_Error_Code := 9011;
    L_Error_Text :=
        'Cluster recovery-lock active';

END_IF;

IF L_Recovery_Valid
   AND L_Cluster_Quarantine THEN

    L_Recovery_Valid := FALSE;

    L_Error_Code := 9012;
    L_Error_Text :=
        'Cluster quarantine active';

END_IF;

IF GVL_SAFETY_RECOVERY.G_Recovery_Active THEN
    GVL_RECOVERY_GOVERNANCE.Recovery_Quarantine_Active := TRUE;
    GVL_RECOVERY_GOVERNANCE.Recovery_Last_Cleanup_Start_MS := L_Now_MS;

    L_Recovery_Valid := FALSE;

    IF L_Error_Code = 0 THEN
        L_Error_Code := 9002;
        L_Error_Text := 'Recovery quarantine active';
    END_IF;
END_IF;

IF L_Recovery_Valid AND GVL_DEGRADED.G_System_Degraded THEN
    L_Recovery_Valid := FALSE;
    L_Error_Code := 9003;
    L_Error_Text := 'Residual degraded state detected';

    GVL_RECOVERY_GOVERNANCE.Recovery_Degraded_State_Residual := TRUE;
END_IF;

IF L_Recovery_Valid AND GVL_TIME_MONOTONIC.Retained_Time_Invalid THEN
    L_Recovery_Valid := FALSE;
    L_Error_Code := 9004;
    L_Error_Text := 'Retained state residue detected';

    GVL_RECOVERY_GOVERNANCE.Recovery_Retained_State_Residual := TRUE;
END_IF;

IF L_Recovery_Valid THEN
    GVL_RECOVERY_GOVERNANCE.Recovery_Epoch := GVL_RECOVERY_GOVERNANCE.Recovery_Epoch + 1;
    GVL_RECOVERY_GOVERNANCE.Recovery_Cleanup_Epoch := GVL_RECOVERY_GOVERNANCE.Recovery_Cleanup_Epoch + 1;

    GVL_RECOVERY_GOVERNANCE.Recovery_Governance_Valid := TRUE;

    // Cleanup release requires finalized publication continuity.
    IF GVL_CONVERGENCE.Convergence_Release_Allowed
       AND L_Finalized_Publication_Continuity THEN

        GVL_RECOVERY_GOVERNANCE.Recovery_Cleanup_Completed := TRUE;
        GVL_RECOVERY_GOVERNANCE.Recovery_Cleanup_Verified := TRUE;
        GVL_RECOVERY_GOVERNANCE.Recovery_Quarantine_Active := FALSE;
        GVL_RECOVERY_GOVERNANCE.Recovery_Forced_Safe_Mode := FALSE;
        GVL_RECOVERY_GOVERNANCE.Recovery_Last_Cleanup_End_MS := L_Now_MS;

        GVL_RECOVERY_GOVERNANCE.Recovery_Last_Error_Code := 0;
        GVL_RECOVERY_GOVERNANCE.Recovery_Last_Error_Text := '';
    ELSE
        GVL_RECOVERY_GOVERNANCE.Recovery_Cleanup_Completed := FALSE;
        GVL_RECOVERY_GOVERNANCE.Recovery_Cleanup_Verified := FALSE;
        GVL_RECOVERY_GOVERNANCE.Recovery_Quarantine_Active := TRUE;
        GVL_RECOVERY_GOVERNANCE.Recovery_Forced_Safe_Mode := TRUE;

        GVL_RECOVERY_GOVERNANCE.Recovery_Last_Error_Code := 9005;
        GVL_RECOVERY_GOVERNANCE.Recovery_Last_Error_Text := 'Recovery cleanup waiting for finalized publication continuity';
    END_IF;
ELSE
    GVL_RECOVERY_GOVERNANCE.Recovery_Governance_Valid := FALSE;
    GVL_RECOVERY_GOVERNANCE.Recovery_Cleanup_Completed := FALSE;
    GVL_RECOVERY_GOVERNANCE.Recovery_Cleanup_Verified := FALSE;

    GVL_RECOVERY_GOVERNANCE.Recovery_Semantic_Residue_Detected := TRUE;
    GVL_RECOVERY_GOVERNANCE.Recovery_Forced_Safe_Mode := TRUE;

    GVL_RECOVERY_GOVERNANCE.Recovery_Last_Error_Code := L_Error_Code;
    GVL_RECOVERY_GOVERNANCE.Recovery_Last_Error_Text := L_Error_Text;

    GVL_RECOVERY_GOVERNANCE.Recovery_Invalidation_Count := GVL_RECOVERY_GOVERNANCE.Recovery_Invalidation_Count + 1;
END_IF;
          
END_PROGRAM

PROGRAM PRG_Presence_Manager
  VAR
    fbPresence : FB_Presence_Manager;
    L_i : INT;
  END_VAR

            fbPresence(
    VI_Motion_Sensors := GVL_STATE.G_Motion_Sensors,
    VI_System_Time_MS := GVL_STATUS.G_System_Time_MS
);

GVL_PRESENCE.G_Any_Motion := fbPresence.VO_Any_Motion;
GVL_PRESENCE.G_Occupied := fbPresence.VO_Occupied;
GVL_PRESENCE.G_Auto_Away_Request := fbPresence.VO_Auto_Away;
GVL_PRESENCE.G_Last_Motion_TS := fbPresence.VO_Last_Motion_TS;

FOR L_i := 1 TO GVL_CONSTANTS.C_MAX_ZONES DO
    IF GVL_STATE.G_Motion_Sensors[L_i] THEN
        GVL_PRESENCE.G_Zone_Occupied[L_i] := TRUE;
        GVL_PRESENCE.G_Zone_Last_Motion_TS[L_i] := GVL_STATUS.G_System_Time_MS;
    END_IF;

    IF (GVL_STATUS.G_System_Time_MS - GVL_PRESENCE.G_Zone_Last_Motion_TS[L_i]) > 900000 THEN
        GVL_PRESENCE.G_Zone_Occupied[L_i] := FALSE;
    END_IF;
END_FOR;
          
END_PROGRAM

PROGRAM PRG_Verification_Domain

            // SEMANTIC DOMAIN WRAPPER

PRG_Passive_Runtime_Verification_Governor();
PRG_Semantic_Drift_Observability_Governor();
PRG_Proof_Continuity_Audit_Governor();
PRG_Runtime_Assumption_Integrity_Governor();

PRG_Command_Verifier();
PRG_Explainability();
          
END_PROGRAM

PROGRAM PRG_Distributed_Snapshot_Ingestion

            // ======================================================
// DISTRIBUTED SNAPSHOT INGESTION
// ======================================================
// Canonical replicated distributed snapshot ingestion.
//
// Purpose:
// normalize replicated immutable snapshot state from
// HA/session replication boundary into peer snapshot fields.
//
// This layer does NOT:
// - perform distributed reconciliation
// - mutate local runtime snapshot authority
// - mutate output/runtime authority
// ======================================================

IF NOT GVL_HA_SESSION_REPLICATION.HA_Remote_Session_Valid THEN
    GVL_DISTRIBUTED_SNAPSHOT.Peer_Distributed_Snapshot_Epoch := 0;
    GVL_DISTRIBUTED_SNAPSHOT.Peer_Runtime_Snapshot_Epoch := 0;
    GVL_DISTRIBUTED_SNAPSHOT.Peer_Publication_Epoch := 0;

    GVL_DISTRIBUTED_SNAPSHOT.Peer_Snapshot_Immutable := FALSE;
    GVL_DISTRIBUTED_SNAPSHOT.Peer_Snapshot_Lease_Active := FALSE;
    GVL_DISTRIBUTED_SNAPSHOT.Peer_Snapshot_Last_Refresh_MS := 0;

    RETURN;
END_IF;

GVL_DISTRIBUTED_SNAPSHOT.Peer_Distributed_Snapshot_Epoch :=
    GVL_HA_SESSION_REPLICATION.HA_Remote_Distributed_Snapshot_Epoch;

GVL_DISTRIBUTED_SNAPSHOT.Peer_Runtime_Snapshot_Epoch :=
    GVL_HA_SESSION_REPLICATION.HA_Remote_Runtime_Snapshot_Epoch;

GVL_DISTRIBUTED_SNAPSHOT.Peer_Publication_Epoch :=
    GVL_HA_SESSION_REPLICATION.HA_Remote_Publication_Epoch;

GVL_DISTRIBUTED_SNAPSHOT.Peer_Snapshot_Immutable :=
    GVL_HA_SESSION_REPLICATION.HA_Remote_Snapshot_Immutable;

GVL_DISTRIBUTED_SNAPSHOT.Peer_Snapshot_Lease_Active := TRUE;

GVL_DISTRIBUTED_SNAPSHOT.Peer_Snapshot_Last_Refresh_MS :=
    GVL_HA_SESSION_REPLICATION.HA_Remote_Snapshot_Last_Refresh_MS;

// >>> BULK_SYNC_ANCHOR: PRG_Distributed_Snapshot_Ingestion <<<
          
END_PROGRAM

PROGRAM PRG_Output_Freshness_Governor
  VAR
    L_Now_MS : UDINT;
    L_Delta_MS : UDINT;
    L_Output_Valid : BOOL := TRUE;
    L_Error_Code : UDINT := 0;
    L_Error_Text : STRING(160) := '';
  END_VAR

            L_Now_MS := GVL_STATUS.G_System_Time_MS;
L_Output_Valid := TRUE;
L_Error_Code := 0;
L_Error_Text := '';

IF NOT GVL_RUNTIME_EPOCH.Runtime_Runtime_Barrier_OK THEN
    L_Output_Valid := FALSE;
    L_Error_Code := 6000;
    L_Error_Text := 'Output runtime authority invalid';
END_IF;

IF L_Output_Valid AND (NOT GVL_RUNTIME_EPOCH.Runtime_IO_Publication_Allowed) THEN
    L_Output_Valid := FALSE;
    L_Error_Code := 6001;
    L_Error_Text := 'Output publication not allowed';
END_IF;

IF L_Output_Valid AND (NOT GVL_RUNTIME_SNAPSHOT.Snapshot_Frozen) THEN
    L_Output_Valid := FALSE;
    L_Error_Code := 6100;
    L_Error_Text := 'Runtime snapshot not frozen';
END_IF;

IF L_Output_Valid AND (NOT GVL_RUNTIME_SNAPSHOT.Snapshot_Publication_Allowed) THEN
    L_Output_Valid := FALSE;
    L_Error_Code := 6101;
    L_Error_Text := 'Snapshot publication blocked';
END_IF;

IF L_Output_Valid AND (NOT GVL_RUNTIME_SNAPSHOT.Snapshot_Copy_Valid) THEN
    L_Output_Valid := FALSE;
    L_Error_Code := 6102;
    L_Error_Text := 'Snapshot copy invalid';
END_IF;

IF L_Output_Valid AND (NOT GVL_RUNTIME_SNAPSHOT.Snapshot_Isolation_Valid) THEN
    L_Output_Valid := FALSE;
    L_Error_Code := 6103;
    L_Error_Text := 'Snapshot isolation invalid';
END_IF;

IF L_Output_Valid AND GVL_RUNTIME_SNAPSHOT.Snapshot_Mutation_Detected THEN
    L_Output_Valid := FALSE;
    L_Error_Code := 6104;
    L_Error_Text := 'Snapshot mutation detected';
END_IF;

IF L_Output_Valid AND GVL_DISTRIBUTED_EPOCH.Distributed_Quarantine_Active THEN
    L_Output_Valid := FALSE;
    L_Error_Code := 6200;
    L_Error_Text := 'Distributed reconciliation quarantine active';
END_IF;

IF L_Output_Valid AND (NOT GVL_DISTRIBUTED_SNAPSHOT.Distributed_Publication_Reconciled) THEN
    L_Output_Valid := FALSE;
    L_Error_Code := 6300;
    L_Error_Text := 'Distributed publication reconciliation invalid';
END_IF;

IF L_Output_Valid AND (NOT GVL_DISTRIBUTED_SNAPSHOT.Distributed_Publication_Freeze_Valid) THEN
    L_Output_Valid := FALSE;
    L_Error_Code := 6301;
    L_Error_Text := 'Distributed publication freeze invalid';
END_IF;

IF L_Output_Valid AND (NOT GVL_DISTRIBUTED_SNAPSHOT.Distributed_Snapshot_Consistent) THEN
    L_Output_Valid := FALSE;
    L_Error_Code := 6302;
    L_Error_Text := 'Distributed immutable snapshot inconsistent';
END_IF;

IF L_Output_Valid AND GVL_DISTRIBUTED_SNAPSHOT.Distributed_Snapshot_Quarantine_Active THEN
    L_Output_Valid := FALSE;
    L_Error_Code := 6306;
    L_Error_Text := 'Distributed immutable snapshot quarantine active';
END_IF;

// Finalized distributed publication continuity.
IF L_Output_Valid AND (NOT GVL_DISTRIBUTED_COMMIT.Distributed_Commit_Valid) THEN
    L_Output_Valid := FALSE;
    L_Error_Code := 6400;
    L_Error_Text := 'Distributed commit invalid';
END_IF;

IF L_Output_Valid AND (NOT GVL_DISTRIBUTED_COMMIT.Publication_Prepare_Valid) THEN
    L_Output_Valid := FALSE;
    L_Error_Code := 6402;
    L_Error_Text := 'Distributed publication prepare invalid';
END_IF;

IF L_Output_Valid AND GVL_DISTRIBUTED_COMMIT.Publication_Commit_Requested
   AND (NOT GVL_DISTRIBUTED_COMMIT.Publication_Commit_Confirmed) THEN
    L_Output_Valid := FALSE;
    L_Error_Code := 6403;
    L_Error_Text := 'Distributed publication commit pending';
END_IF;

IF L_Output_Valid AND GVL_DISTRIBUTED_COMMIT.Peer_Commit_Mismatch THEN
    L_Output_Valid := FALSE;
    L_Error_Code := 6404;
    L_Error_Text := 'Distributed peer commit mismatch';
END_IF;

IF L_Output_Valid AND GVL_DISTRIBUTED_COMMIT.Distributed_Commit_Quarantine_Active THEN
    L_Output_Valid := FALSE;
    L_Error_Code := 6401;
    L_Error_Text := 'Distributed commit quarantine active';
END_IF;

IF L_Output_Valid AND GVL_DISTRIBUTED_COMMIT.Commit_Lease_Expired THEN
    L_Output_Valid := FALSE;
    L_Error_Code := 6405;
    L_Error_Text := 'Distributed commit lease expired';
END_IF;

GVL_OUTPUT_EPOCH.Output_Semantic_Continuity_Warning :=
    (NOT GVL_SEMANTIC_PROGRESS.Semantic_Forward_Progress_Valid)
    OR (NOT GVL_SEMANTIC_PROGRESS.Semantic_Execution_Continuity_OK)
    OR GVL_SEMANTIC_PROGRESS.Semantic_Stagnation_Detected
    OR GVL_SEMANTIC_PROGRESS.Semantic_Replay_Suspected
    OR GVL_SEMANTIC_PROGRESS.Semantic_Livelock_Suspected
    OR GVL_SEMANTIC_PROGRESS.Semantic_Deadlock_Suspected
    OR GVL_SEMANTIC_PROGRESS.Semantic_Progress_Lease_Expired
    OR GVL_SEMANTIC_PROGRESS.Semantic_Progress_Quarantine_Active;

// Hard semantic continuity invalidation.
IF L_Output_Valid
AND GVL_OUTPUT_EPOCH.Output_Semantic_Continuity_Warning
THEN
    L_Output_Valid := FALSE;
    L_Error_Code := 6500;
    L_Error_Text := 'Semantic continuity invalid';
END_IF;

IF L_Output_Valid THEN
    IF GVL_OUTPUT_EPOCH.Output_Runtime_Epoch > GVL_RUNTIME_EPOCH.Runtime_Epoch THEN
        L_Output_Valid := FALSE;
        L_Error_Code := 6002;
        L_Error_Text := 'Output epoch ahead of runtime epoch';
    END_IF;
END_IF;

L_Delta_MS := L_Now_MS - GVL_OUTPUT_EPOCH.Output_Last_Refresh_MS;

IF L_Output_Valid AND GVL_OUTPUT_EPOCH.Output_Lease_Active THEN
    IF L_Delta_MS > GVL_OUTPUT_EPOCH.Output_Lease_Timeout_MS THEN
        L_Output_Valid := FALSE;
        L_Error_Code := 6003;
        L_Error_Text := 'Output lease expired';
    END_IF;
END_IF;

IF L_Output_Valid THEN
    GVL_OUTPUT_EPOCH.Output_Publication_Epoch := GVL_OUTPUT_EPOCH.Output_Publication_Epoch + 1;

    GVL_OUTPUT_EPOCH.Output_Publication_Valid := TRUE;
    GVL_OUTPUT_EPOCH.Output_Lease_Active := TRUE;
    GVL_OUTPUT_EPOCH.Output_Lease_Expired := FALSE;

    GVL_OUTPUT_EPOCH.Output_Runtime_Epoch := GVL_RUNTIME_EPOCH.Runtime_Epoch;
    GVL_OUTPUT_EPOCH.Output_Runtime_Epoch_Valid := TRUE;

    GVL_OUTPUT_EPOCH.Output_Last_Publication_MS := L_Now_MS;
    GVL_OUTPUT_EPOCH.Output_Last_Refresh_MS := L_Now_MS;

    IF GVL_CONVERGENCE.Convergence_Release_Allowed THEN
        GVL_OUTPUT_EPOCH.Output_Stale_Detected := FALSE;
        GVL_OUTPUT_EPOCH.Output_Forced_Safe_Decay := FALSE;
    END_IF;

    GVL_OUTPUT_EPOCH.Output_Last_Error_Code := 0;
    GVL_OUTPUT_EPOCH.Output_Last_Error_Text := '';
ELSE
    GVL_OUTPUT_EPOCH.Output_Publication_Valid := FALSE;
    GVL_OUTPUT_EPOCH.Output_Lease_Expired := TRUE;
    GVL_OUTPUT_EPOCH.Output_Stale_Detected := TRUE;
    GVL_OUTPUT_EPOCH.Output_Forced_Safe_Decay := TRUE;

    GVL_OUTPUT_EPOCH.Output_Last_Invalidation_MS := L_Now_MS;
    GVL_OUTPUT_EPOCH.Output_Last_Error_Code := L_Error_Code;
    GVL_OUTPUT_EPOCH.Output_Last_Error_Text := L_Error_Text;
END_IF;
          
END_PROGRAM

PROGRAM PRG_Policy

            // ============================================================
// CONFIGURATION SAFETY CLAMP
// ============================================================
// Configuration validation is diagnostic-only here.
// System mode ownership remains in FB_State_Manager via
// FB_System_Health_Orchestrator. Policy must not directly write
// GVL_STATE.G_System_Mode.
IF GVL_CONFIG_VALIDATION.G_Config_Force_Safe_Mode AND
   (NOT GVL_CONFIG_VALIDATION.G_Config_Valid) AND
   (GVL_STATE.G_System_Mode = E_System_Operating_Mode.MODE_NORMAL) THEN
    GVL_STATUS.G_Diagnostics.Subsystem_Degraded := TRUE;
    GVL_STATUS.G_System_Mode_Text := 'CONFIG DEGRADED';
END_IF;

// ============================================================
// SCENARIO POLICY OWNER
// ============================================================

// 1. Base priority resolution
IF GVL_STATE.G_System_Mode = E_System_Operating_Mode.MODE_SAFE_STOP THEN
    GVL_POLICY.G_Scenario_Intent := E_SCENARIO_TYPE.SCENARIO_NONE;
    GVL_POLICY.G_Scenario_Source := SRC_SAFETY;

ELSIF GVL_POLICY.G_Scenario_Request_Operator <> E_SCENARIO_TYPE.SCENARIO_NONE THEN
    GVL_POLICY.G_Scenario_Intent := GVL_POLICY.G_Scenario_Request_Operator;
    GVL_POLICY.G_Scenario_Source := SRC_OPERATOR;

ELSIF GVL_POLICY.G_Scenario_Request_Gateway <> E_SCENARIO_TYPE.SCENARIO_NONE THEN
    GVL_POLICY.G_Scenario_Intent := GVL_POLICY.G_Scenario_Request_Gateway;
    GVL_POLICY.G_Scenario_Source := SRC_GATEWAY;

ELSIF GVL_POLICY.G_Scenario_Request_Rule <> E_SCENARIO_TYPE.SCENARIO_NONE THEN
    GVL_POLICY.G_Scenario_Intent := GVL_POLICY.G_Scenario_Request_Rule;
    GVL_POLICY.G_Scenario_Source := SRC_RULE;

ELSE
    GVL_POLICY.G_Scenario_Intent := GVL_STATUS.G_Current_Scenario;
    GVL_POLICY.G_Scenario_Source := SRC_NONE;
END_IF;

// 2. Fail-safe clamp
CASE GVL_STATE.G_System_Mode OF
    E_System_Operating_Mode.MODE_SAFE_STOP:
        GVL_POLICY.G_Scenario_Intent := E_SCENARIO_TYPE.SCENARIO_NONE;
        GVL_POLICY.G_Scenario_Source := SRC_SAFETY;

    E_System_Operating_Mode.MODE_FREEZE_PROTECTION:
        GVL_POLICY.G_Scenario_Intent := E_SCENARIO_TYPE.SCENARIO_NONE;
        GVL_POLICY.G_Scenario_Source := SRC_POLICY;

    E_System_Operating_Mode.MODE_DEGRADED:
        CASE GVL_POLICY.G_Scenario_Intent OF
            E_SCENARIO_TYPE.SCENARIO_NONE,
            E_SCENARIO_TYPE.SCENARIO_PRESENCE,
            E_SCENARIO_TYPE.SCENARIO_AWAY,
            E_SCENARIO_TYPE.SCENARIO_SLEEP:
                ;
        ELSE
            GVL_POLICY.G_Scenario_Intent := E_SCENARIO_TYPE.SCENARIO_NONE;
            GVL_POLICY.G_Scenario_Source := SRC_POLICY;
        END_CASE;
END_CASE;

// 3. Context automation
IF GVL_STATE.G_System_Mode = E_System_Operating_Mode.MODE_NORMAL THEN
    IF GVL_ALARM.G_Security_Armed AND
       (GVL_POLICY.G_Scenario_Request_Operator = E_SCENARIO_TYPE.SCENARIO_NONE) AND
       (GVL_POLICY.G_Scenario_Request_Gateway = E_SCENARIO_TYPE.SCENARIO_NONE) AND
       (GVL_POLICY.G_Scenario_Request_Rule = E_SCENARIO_TYPE.SCENARIO_NONE) AND
       (GVL_POLICY.G_Scenario_Intent <> E_SCENARIO_TYPE.SCENARIO_AWAY) THEN
        GVL_POLICY.G_Scenario_Intent := E_SCENARIO_TYPE.SCENARIO_AWAY;
        GVL_POLICY.G_Scenario_Source := SRC_POLICY;
    END_IF;
END_IF;

// 4. Degraded adaptation
IF GVL_STATE.G_System_Mode = E_System_Operating_Mode.MODE_DEGRADED THEN
    IF (GVL_POLICY.G_Scenario_Request_Operator = E_SCENARIO_TYPE.SCENARIO_NONE) AND
       (GVL_POLICY.G_Scenario_Request_Gateway = E_SCENARIO_TYPE.SCENARIO_NONE) AND
       (GVL_POLICY.G_Scenario_Request_Rule = E_SCENARIO_TYPE.SCENARIO_NONE) THEN

        IF GVL_ALARM.G_Security_Armed THEN
            GVL_POLICY.G_Scenario_Intent := E_SCENARIO_TYPE.SCENARIO_AWAY;
            GVL_POLICY.G_Scenario_Source := SRC_POLICY;

        ELSIF GVL_POLICY.G_Scenario_Intent = E_SCENARIO_TYPE.SCENARIO_PRESENCE THEN
            GVL_POLICY.G_Scenario_Intent := E_SCENARIO_TYPE.SCENARIO_SLEEP;
            GVL_POLICY.G_Scenario_Source := SRC_POLICY;
        END_IF;
    END_IF;
END_IF;

// 5. Heating bridge
GVL_STATE.G_Preheat_Request := GVL_POLICY.G_Rule_Preheat_Request;
GVL_STATE.G_Freeze_Request :=
    (GVL_STATE.G_System_Mode = E_System_Operating_Mode.MODE_FREEZE_PROTECTION);
          
END_PROGRAM

PROGRAM PRG_Water_Supervisory_Publication
  VAR
    fbConfigActivationRuntime : FB_Config_Activation_Runtime;
    fbHMIConfigWorkflowRuntime : FB_HMI_Config_Workflow_Runtime;
    fbRestartContinuity : FB_Runtime_Restart_Continuity;
    fbWaterHardwareBindingRuntime : FB_Water_Hardware_Binding_Runtime;
    fbWaterTopologyConfig : FB_Water_Topology_Config_Runtime;
    fbWaterLeakProjection : FB_Water_Leak_Runtime_Projection;
    fbWaterTopologyValidator : FB_Water_Hydraulic_Topology_Validator;
    fbWaterIsolationPathResolver : FB_Water_Isolation_Path_Resolver;
    fbWaterOrchestrationRuntime : FB_Water_Orchestration_Runtime;
    fbWaterIsolationProjection : FB_Water_Isolation_Runtime_Projection;
    fbWaterIsolationIntentBuilder : FB_Water_Isolation_Intent_Builder;
    fbWaterAuthorityArbitrator : FB_Water_Isolation_Authority_Arbitrator;
    fbWaterValveGovernance : FB_Water_Valve_Runtime_Governance;
    L_i : INT;
    L_State : ST_Water_Leak_Runtime_State;
    L_Any_Leak : BOOL;
    L_Any_Warning : BOOL;
    L_Any_Degraded_Mapping : BOOL;
    L_Selective_Isolation_Available : BOOL;
    L_Global_Fallback_Required : BOOL;
  END_VAR

            // Water/Flood supervisory publication orchestration.
//
// Runtime chain:
// config activation/workflow
//   -> restart continuity
//   -> hardware binding resolver
//   -> runtime topology config
//   -> leak semantics
//   -> topology validation
//   -> graph/path resolution
//   -> orchestration/traversal governance
//   -> isolation semantics
//   -> authority arbitration
//   -> valve governance
//   -> supervisory publication
//
// Distributed execution gates are authoritative.
// Water runtime orchestration must never bypass cluster execution policy.

fbConfigActivationRuntime(
    VI_Enable := TRUE,
    VI_System_Time_MS := GVL_STATUS.G_System_Time_MS
);

fbHMIConfigWorkflowRuntime(
    VI_Enable := TRUE,
    VI_System_Time_MS := GVL_STATUS.G_System_Time_MS
);

fbRestartContinuity(
    VI_Enable := TRUE,
    VI_System_Time_MS := GVL_STATUS.G_System_Time_MS,
    VI_Warm_Restart := GVL_Runtime_Restart_Continuity.G_Restore_Request
);

fbWaterHardwareBindingRuntime(
    VI_Enable := TRUE,
    VI_System_Time_MS := GVL_STATUS.G_System_Time_MS
);

fbWaterTopologyConfig(
    VI_Enable := TRUE,
    VI_System_Time_MS := GVL_STATUS.G_System_Time_MS
);

fbWaterLeakProjection(
    VI_Enable := TRUE,
    VI_System_Time_MS := GVL_STATUS.G_System_Time_MS
);

fbWaterTopologyValidator(
    VI_Enable := TRUE,
    VI_System_Time_MS := GVL_STATUS.G_System_Time_MS
);

fbWaterIsolationPathResolver(
    VI_Enable := GVL_Distributed_Execution_Gates.G_Can_Orchestrate,
    VI_System_Time_MS := GVL_STATUS.G_System_Time_MS
);

fbWaterOrchestrationRuntime(
    VI_Enable := GVL_Distributed_Execution_Gates.G_Can_Orchestrate,
    VI_System_Time_MS := GVL_STATUS.G_System_Time_MS
);

fbWaterIsolationProjection(
    VI_Enable := GVL_Distributed_Execution_Gates.G_Can_Execute,
    VI_System_Time_MS := GVL_STATUS.G_System_Time_MS
);

fbWaterIsolationIntentBuilder(
    VI_Enable := GVL_Distributed_Execution_Gates.G_Can_Execute
);

fbWaterAuthorityArbitrator(
    VI_Enable := GVL_Distributed_Execution_Gates.G_Can_Execute,
    VI_System_Time_MS := GVL_STATUS.G_System_Time_MS
);

fbWaterValveGovernance(
    VI_Enable := GVL_Distributed_Execution_Gates.G_Can_Own_Projection,
    VI_System_Time_MS := GVL_STATUS.G_System_Time_MS
);

L_Any_Leak := FALSE;
L_Any_Warning := FALSE;
L_Any_Degraded_Mapping := FALSE;
L_Selective_Isolation_Available := FALSE;
L_Global_Fallback_Required := FALSE;

FOR L_i := 1 TO GVL_CONSTANTS.C_MAX_FLOOD_SENSORS DO

    L_State := GVL_Water_Runtime_Projection.G_Leak_Runtime_State[L_i];

    L_Any_Leak := L_Any_Leak OR L_State.Leak_Confirmed;
    L_Any_Warning := L_Any_Warning OR L_State.Leak_Warning_Active;

    L_Any_Degraded_Mapping :=
        L_Any_Degraded_Mapping
        OR GVL_Water_Orchestration.G_Traversal_State[L_i].Traversal_Conflict
        OR NOT GVL_Water_Topology_Config.G_Config_Record[L_i].Config_Valid
        OR GVL_IO_Binding_Runtime.G_Any_Invalid_Binding;

    L_Selective_Isolation_Available :=
        L_Selective_Isolation_Available
        OR GVL_Water_Orchestration.G_Traversal_State[L_i].Selective_Path_Allowed;

    L_Global_Fallback_Required :=
        L_Global_Fallback_Required
        OR GVL_Water_Orchestration.G_Traversal_State[L_i].Global_Fallback_Required;

END_FOR;

GVL_Water_Runtime_Supervisory_Publication.G_Supervisory_Valid := TRUE;
GVL_Water_Runtime_Supervisory_Publication.G_Last_Update_MS :=
    GVL_STATUS.G_System_Time_MS;

GVL_Water_Runtime_Supervisory_Publication.G_Any_Leak_Active :=
    L_Any_Leak;

GVL_Water_Runtime_Supervisory_Publication.G_Any_Warning_Active :=
    L_Any_Warning;

GVL_Water_Runtime_Supervisory_Publication.G_Any_Degraded_Mapping :=
    L_Any_Degraded_Mapping;

GVL_Water_Runtime_Supervisory_Publication.G_Selective_Isolation_Available :=
    L_Selective_Isolation_Available;

GVL_Water_Runtime_Supervisory_Publication.G_Global_Fallback_Active :=
    L_Global_Fallback_Required;

IF NOT GVL_Distributed_Execution_Gates.G_Can_Execute THEN
    GVL_Water_Runtime_Supervisory_Publication.G_Status_Code := 20;
    GVL_Water_Runtime_Supervisory_Publication.G_Status_Text :=
        'Distributed execution gates restricted';
ELSIF GVL_Config_Activation.G_Config_Quarantine_Active THEN
    GVL_Water_Runtime_Supervisory_Publication.G_Status_Code := 11;
    GVL_Water_Runtime_Supervisory_Publication.G_Status_Text :=
        'Runtime config quarantine active';
ELSIF GVL_IO_Binding_Runtime.G_Any_Invalid_Binding THEN
    GVL_Water_Runtime_Supervisory_Publication.G_Status_Code := 10;
    GVL_Water_Runtime_Supervisory_Publication.G_Status_Text :=
        'Hardware binding invalid';
ELSIF GVL_Water_Topology_Config.G_Any_Invalid_Config THEN
    GVL_Water_Runtime_Supervisory_Publication.G_Status_Code := 8;
    GVL_Water_Runtime_Supervisory_Publication.G_Status_Text :=
        'Runtime topology config invalid';
ELSIF GVL_Water_Orchestration.G_Any_Escalation_Required THEN
    GVL_Water_Runtime_Supervisory_Publication.G_Status_Code := 7;
    GVL_Water_Runtime_Supervisory_Publication.G_Status_Text :=
        'Topology-aware orchestration escalation active';
ELSIF GVL_Water_Orchestration.G_Any_Traversal_Conflict THEN
    GVL_Water_Runtime_Supervisory_Publication.G_Status_Code := 6;
    GVL_Water_Runtime_Supervisory_Publication.G_Status_Text :=
        'Traversal conflict detected';
ELSE
    GVL_Water_Runtime_Supervisory_Publication.G_Status_Code := 0;
    GVL_Water_Runtime_Supervisory_Publication.G_Status_Text :=
        'Runtime topology orchestration active';
END_IF;

// >>> BULK_SYNC_ANCHOR: PRG_Water_Supervisory_Publication <<<
          
END_PROGRAM

PROGRAM PRG_Safety_Shutdown
  VAR
    L_Mode : E_Safety_Mode := NORMAL;
  END_VAR

            // Input degraded forces safe stop first
IF GVL_INPUT.IN_Input_Degraded THEN
    L_Mode := GLOBAL_STOP;
ELSE

    // Priority: FIRE > GAS > WATER > GLOBAL_STOP > NORMAL

    IF GVL_INTENT_SAFETY.I_Fire_Alarm_Active THEN
        L_Mode := FIRE;
    ELSIF GVL_INTENT_SAFETY.I_Gas_Close_Required OR GVL_INTENT_SAFETY.I_Test_Timeout_Gas_Close THEN
        L_Mode := GAS;
    ELSIF GVL_INTENT_SAFETY.I_Water_Main_Close_Required OR GVL_INTENT_SAFETY.I_Test_Timeout_Water_Close THEN
        L_Mode := WATER_LEAK;
    ELSIF GVL_INTENT_SAFETY.I_System_Safe_Stop_Required THEN
        L_Mode := GLOBAL_STOP;
    ELSE
        L_Mode := NORMAL;
    END_IF;

END_IF;

GVL_SAFETY_SHUTDOWN.G_Safety_Mode := L_Mode;
GVL_SAFETY_SHUTDOWN.G_Safety_Active := (L_Mode <> NORMAL);

// >>> BULK_SYNC_ANCHOR: PRG_Safety_Shutdown <<<
          
END_PROGRAM

PROGRAM PRG_IO_Write
  VAR
    L_i : INT;
    L_Heating_Forced_Off : BOOL;
    L_Vent_Forced_Off : BOOL;
    L_Water_Forced_Off : BOOL;
    L_Access_Forced_Off : BOOL;
    L_Access_Safety_Override : BOOL;
    L_Global_Hard_Stop : BOOL;
    L_Gas_Safety_Stop : BOOL;
    L_Freeze_Active : BOOL;
    L_Gas_Fire_Siren_Enable : BOOL;
    L_PreOutput_Block_IO : BOOL;
    L_Output_Freshness_Block : BOOL;
    L_Output_Publication_Block : BOOL;
    L_Distributed_Publication_Block : BOOL;
    L_Snapshot_Block : BOOL;
    L_Distributed_Execution_Block : BOOL;
    L_Gas_Siren_Authority : BOOL;
    L_Fire_Siren_Authority : BOOL;
    fbTrace : FB_Trace_Write;
  END_VAR

            L_PreOutput_Block_IO := GVL_COMMAND_VERIFY.PreOutput_Block_IO;
L_Output_Freshness_Block := GVL_OUTPUT_EPOCH.Output_Forced_Safe_Decay;

L_Output_Publication_Block :=
    (NOT GVL_OUTPUT_EPOCH.Output_Publication_Valid)
    OR (NOT GVL_OUTPUT_EPOCH.Output_Runtime_Epoch_Valid)
    OR GVL_OUTPUT_EPOCH.Output_Lease_Expired;

// Final distributed publication continuity authority.
L_Distributed_Publication_Block :=
    (NOT GVL_DISTRIBUTED_COMMIT.Distributed_Commit_Valid)
    OR GVL_DISTRIBUTED_COMMIT.Distributed_Commit_Quarantine_Active
    OR GVL_DISTRIBUTED_COMMIT.Commit_Lease_Expired
    OR (NOT GVL_DISTRIBUTED_SNAPSHOT.Distributed_Publication_Reconciled)
    OR (NOT GVL_DISTRIBUTED_SNAPSHOT.Distributed_Publication_Freeze_Valid)
    OR (NOT GVL_DISTRIBUTED_SNAPSHOT.Distributed_Snapshot_Consistent);

L_Snapshot_Block :=
    (NOT GVL_RUNTIME_SNAPSHOT.Snapshot_Frozen)
    OR (NOT GVL_RUNTIME_SNAPSHOT.Snapshot_Publication_Allowed)
    OR (NOT GVL_RUNTIME_SNAPSHOT.Snapshot_Copy_Valid)
    OR (NOT GVL_RUNTIME_SNAPSHOT.Snapshot_Isolation_Valid)
    OR GVL_RUNTIME_SNAPSHOT.Snapshot_Mutation_Detected;

L_Distributed_Execution_Block :=
    NOT GVL_Distributed_Execution_Gates.G_Can_Execute
    OR NOT GVL_Distributed_Execution_Gates.G_Can_Own_Projection;

L_Global_Hard_Stop :=
    GVL_COMMAND_SHADOW.G_Heating_Emergency_Stop
    OR L_PreOutput_Block_IO
    OR L_Output_Freshness_Block
    OR L_Output_Publication_Block
    OR L_Distributed_Publication_Block
    OR L_Snapshot_Block
    OR L_Distributed_Execution_Block;

L_Gas_Safety_Stop := GVL_COMMAND_SHADOW.G_Heating_Gas_Safety_Stop OR GVL_COMMAND_SHADOW.G_Boiler_Stop;
L_Freeze_Active := GVL_STATE.G_Safety_Freeze_Risk;
L_Gas_Fire_Siren_Enable := GVL_ALARM.G_Gas_Fire_Siren OR GVL_ALARM.G_Global_Siren OR GVL_ALARM.G_Global_Critical;

L_Gas_Siren_Authority := GVL_HEALTH_BRIDGE.G_Gas_Detected OR GVL_HEALTH_BRIDGE.G_CO_Alarm_Level OR GVL_STATE.G_Safety_Gas_Latched;
L_Fire_Siren_Authority := GVL_HEALTH_BRIDGE.G_Smoke_Detected OR GVL_STATE.G_Safety_Smoke_Latched;

IF NOT GVL_STATUS.G_Is_Active_PLC OR L_Global_Hard_Stop THEN

    FOR L_i := 1 TO GVL_CONSTANTS.C_MAX_HEATING_CIRCUITS DO
        GVL_IO.DO_Zone_Valves[L_i] := FALSE;
    END_FOR;

    GVL_IO.DO_Gas_Valve_Close := TRUE;

    IF L_Distributed_Publication_Block THEN
        fbTrace(
            iLayer := TRACE_IO,
            iSource := SRC_IO,
            iReason := REASON_SAFETY_BLOCK,
            iValueBool := TRUE,
            iValueReal := UDINT_TO_REAL(GVL_DISTRIBUTED_COMMIT.Distributed_Commit_Last_Error_Code),
            iText := 'IO blocked by distributed publication continuity authority');
    END_IF;

    IF L_Output_Publication_Block THEN
        fbTrace(
            iLayer := TRACE_IO,
            iSource := SRC_IO,
            iReason := REASON_SAFETY_BLOCK,
            iValueBool := TRUE,
            iValueReal := UDINT_TO_REAL(GVL_OUTPUT_EPOCH.Output_Last_Error_Code),
            iText := 'IO blocked by finalized output publication authority');
    END_IF;

    RETURN;
END_IF;

fbTrace(
    iLayer := TRACE_IO,
    iSource := SRC_IO,
    iReason := REASON_DOMAIN_PROJECTION,
    iValueBool := TRUE,
    iValueReal := 0.0,
    iText := 'IO write projection executed');
          
END_PROGRAM

PROGRAM PRG_Actuator_Semantic_Verification_Governor
  VAR
    L_Now_MS : UDINT;
    L_Actuator_Valid : BOOL := TRUE;
    L_Error_Code : UDINT := 0;
    L_Error_Text : STRING(160) := '';
  END_VAR

            L_Now_MS := GVL_STATUS.G_System_Time_MS;
L_Actuator_Valid := TRUE;
L_Error_Code := 0;
L_Error_Text := '';

// Fail-safe defaults.
GVL_ACTUATOR_SEMANTIC_VERIFICATION.Actuator_Semantic_Verification_Valid := FALSE;
GVL_ACTUATOR_SEMANTIC_VERIFICATION.Actuator_Semantic_Verification_Granted := FALSE;
GVL_ACTUATOR_SEMANTIC_VERIFICATION.Actuator_Semantic_Verification_Quarantine_Active := TRUE;

GVL_ACTUATOR_SEMANTIC_VERIFICATION.Valve_Semantic_Realization_Valid := FALSE;
GVL_ACTUATOR_SEMANTIC_VERIFICATION.Relay_Semantic_Realization_Valid := FALSE;
GVL_ACTUATOR_SEMANTIC_VERIFICATION.Pump_Semantic_Realization_Valid := FALSE;
GVL_ACTUATOR_SEMANTIC_VERIFICATION.Fan_Semantic_Realization_Valid := FALSE;
GVL_ACTUATOR_SEMANTIC_VERIFICATION.Hydraulic_Response_Valid := FALSE;

// Control temporal coherence required.
IF NOT GVL_CONTROL_TIMING_FABRIC.Control_Temporal_Coherence_Granted THEN
    L_Actuator_Valid := FALSE;
    L_Error_Code := 36000;
    L_Error_Text := 'Control temporal coherence not granted';
END_IF;

// Semantic realization failure detectors.
IF GVL_ACTUATOR_SEMANTIC_VERIFICATION.False_Positive_Actuation_Detected THEN
    L_Actuator_Valid := FALSE;
    L_Error_Code := 36001;
    L_Error_Text := 'False-positive actuation detected';
END_IF;

IF GVL_ACTUATOR_SEMANTIC_VERIFICATION.Mechanical_NonRealization_Detected THEN
    L_Actuator_Valid := FALSE;
    L_Error_Code := 36002;
    L_Error_Text := 'Mechanical non-realization detected';
END_IF;

IF GVL_ACTUATOR_SEMANTIC_VERIFICATION.Welded_Relay_Semantics_Detected THEN
    L_Actuator_Valid := FALSE;
    L_Error_Code := 36003;
    L_Error_Text := 'Welded relay semantics detected';
END_IF;

IF GVL_ACTUATOR_SEMANTIC_VERIFICATION.Hydraulic_NoEffect_Execution_Detected THEN
    L_Actuator_Valid := FALSE;
    L_Error_Code := 36004;
    L_Error_Text := 'Hydraulic no-effect execution detected';
END_IF;

IF GVL_ACTUATOR_SEMANTIC_VERIFICATION.Airflow_Realization_Mismatch_Detected THEN
    L_Actuator_Valid := FALSE;
    L_Error_Code := 36005;
    L_Error_Text := 'Airflow realization mismatch detected';
END_IF;

IF GVL_ACTUATOR_SEMANTIC_VERIFICATION.Physical_Convergence_Divergence_Detected THEN
    L_Actuator_Valid := FALSE;
    L_Error_Code := 36006;
    L_Error_Text := 'Physical convergence divergence detected';
END_IF;

// Physical semantic convergence validation.
IF L_Actuator_Valid
AND NOT GVL_ACTUATOR_SEMANTIC_VERIFICATION.Physical_Effect_Converged THEN
    L_Actuator_Valid := FALSE;
    L_Error_Code := 36010;
    L_Error_Text := 'Physical effect convergence invalid';
END_IF;

IF L_Actuator_Valid
AND NOT GVL_ACTUATOR_SEMANTIC_VERIFICATION.Actuation_Response_Temporal_Valid THEN
    L_Actuator_Valid := FALSE;
    L_Error_Code := 36011;
    L_Error_Text := 'Actuation response timing invalid';
END_IF;

IF L_Actuator_Valid
AND NOT GVL_ACTUATOR_SEMANTIC_VERIFICATION.Sensor_Confirmed_Execution_Valid THEN
    L_Actuator_Valid := FALSE;
    L_Error_Code := 36012;
    L_Error_Text := 'Sensor-confirmed execution invalid';
END_IF;

IF L_Actuator_Valid
AND NOT GVL_ACTUATOR_SEMANTIC_VERIFICATION.Semantic_Outcome_Aligned THEN
    L_Actuator_Valid := FALSE;
    L_Error_Code := 36013;
    L_Error_Text := 'Semantic outcome alignment invalid';
END_IF;

IF L_Actuator_Valid THEN
    GVL_ACTUATOR_SEMANTIC_VERIFICATION.Actuator_Semantic_Verification_Valid := TRUE;
    GVL_ACTUATOR_SEMANTIC_VERIFICATION.Actuator_Semantic_Verification_Granted := TRUE;
    GVL_ACTUATOR_SEMANTIC_VERIFICATION.Actuator_Semantic_Verification_Quarantine_Active := FALSE;

    GVL_ACTUATOR_SEMANTIC_VERIFICATION.Valve_Semantic_Realization_Valid := TRUE;
    GVL_ACTUATOR_SEMANTIC_VERIFICATION.Relay_Semantic_Realization_Valid := TRUE;
    GVL_ACTUATOR_SEMANTIC_VERIFICATION.Pump_Semantic_Realization_Valid := TRUE;
    GVL_ACTUATOR_SEMANTIC_VERIFICATION.Fan_Semantic_Realization_Valid := TRUE;
    GVL_ACTUATOR_SEMANTIC_VERIFICATION.Hydraulic_Response_Valid := TRUE;

    GVL_ACTUATOR_SEMANTIC_VERIFICATION.Actuator_Verification_Epoch :=
        GVL_CONTROL_TIMING_FABRIC.Control_Timing_Epoch;

    GVL_ACTUATOR_SEMANTIC_VERIFICATION.Actuator_Verification_Epoch_Coherent := TRUE;

    GVL_ACTUATOR_SEMANTIC_VERIFICATION.Actuator_Verification_Last_Update_MS :=
        L_Now_MS;

    GVL_ACTUATOR_SEMANTIC_VERIFICATION.Actuator_Verification_Lease_Expired := FALSE;

    GVL_ACTUATOR_SEMANTIC_VERIFICATION.Actuator_Verification_Last_Error_Code := 0;
    GVL_ACTUATOR_SEMANTIC_VERIFICATION.Actuator_Verification_Last_Error_Text := '';
ELSE
    GVL_ACTUATOR_SEMANTIC_VERIFICATION.Actuator_Semantic_Verification_Valid := FALSE;
    GVL_ACTUATOR_SEMANTIC_VERIFICATION.Actuator_Semantic_Verification_Granted := FALSE;
    GVL_ACTUATOR_SEMANTIC_VERIFICATION.Actuator_Semantic_Verification_Quarantine_Active := TRUE;

    GVL_ACTUATOR_SEMANTIC_VERIFICATION.Actuator_Verification_Lease_Expired := TRUE;

    GVL_ACTUATOR_SEMANTIC_VERIFICATION.Actuator_Verification_Last_Error_Code :=
        L_Error_Code;

    GVL_ACTUATOR_SEMANTIC_VERIFICATION.Actuator_Verification_Last_Error_Text :=
        L_Error_Text;

    GVL_ACTUATOR_SEMANTIC_VERIFICATION.Actuator_Verification_Invalidation_Count :=
        GVL_ACTUATOR_SEMANTIC_VERIFICATION.Actuator_Verification_Invalidation_Count + 1;
END_IF;
          
END_PROGRAM

PROGRAM PRG_System_History
  VAR
    fbHistoryManager : FB_History_Manager;
    L_History_Event : ST_History_Record;
    L_History_Write_Event : BOOL;
    L_Last_System_Mode : E_System_Operating_Mode;
    L_Last_Root_Cause : E_System_Root_Cause;
    L_Last_First_Fault_Source : INT;
    L_Last_Operator_Journal_Seq : UDINT;
    L_Last_Event_Code : UDINT;
    L_Last_Event_Value : REAL;
    L_Last_Event_Time_MS : UDINT;
  END_VAR

            L_History_Write_Event := FALSE;
L_History_Event.timestamp_ms := GVL_TIME_SERVICE.G_Now_MS;
L_History_Event.event_code := 0;
L_History_Event.event_value := 0.0;
L_History_Event.unit := 0;
L_History_Event.zone_id := 0;
L_History_Event.operator_id := 'SYSTEM';
L_History_Event.priority := E_ALERT_PRIORITY.ALERT_PRIORITY_HIGH;

IF GVL_STATE.G_System_Mode <> L_Last_System_Mode THEN
    L_History_Write_Event := TRUE;
    L_History_Event.event_code := 1101;
    L_History_Event.event_value := TO_REAL(TO_INT(GVL_STATE.G_System_Mode));
    L_History_Event.unit := 1;
    L_History_Event.zone_id := 0;
    L_History_Event.priority := E_ALERT_PRIORITY.ALERT_PRIORITY_HIGH;
    L_Last_System_Mode := GVL_STATE.G_System_Mode;

ELSIF GVL_SYSTEM_HEALTH.G_Root_Cause <> L_Last_Root_Cause THEN
    L_History_Write_Event := TRUE;
    L_History_Event.event_code := 1102;
    L_History_Event.event_value := TO_REAL(TO_INT(GVL_SYSTEM_HEALTH.G_Root_Cause));
    L_History_Event.unit := 2;
    L_History_Event.zone_id := TO_BYTE(GVL_SYSTEM_HEALTH.G_First_Fault_Source);
    L_History_Event.priority := E_ALERT_PRIORITY.ALERT_PRIORITY_HIGH;
    L_Last_Root_Cause := GVL_SYSTEM_HEALTH.G_Root_Cause;

ELSIF GVL_SYSTEM_HEALTH.G_First_Fault_Source <> L_Last_First_Fault_Source THEN
    L_History_Write_Event := TRUE;
    L_History_Event.event_code := 1103;
    L_History_Event.event_value := TO_REAL(GVL_SYSTEM_HEALTH.G_First_Fault_Source);
    L_History_Event.unit := 3;
    L_History_Event.zone_id := TO_BYTE(GVL_SYSTEM_HEALTH.G_First_Fault_Source);
    L_History_Event.priority := E_ALERT_PRIORITY.ALERT_PRIORITY_HIGH;
    L_Last_First_Fault_Source := GVL_SYSTEM_HEALTH.G_First_Fault_Source;

ELSIF GVL_STATUS.G_Current_Scenario <> GVL_STATUS.G_Previous_Scenario THEN
    L_History_Write_Event := TRUE;
    L_History_Event.event_code := 1001;
    L_History_Event.event_value := TO_REAL(GVL_STATUS.G_Current_Scenario);
    L_History_Event.unit := 4;
    L_History_Event.zone_id := 0;
    L_History_Event.priority := E_ALERT_PRIORITY.ALERT_PRIORITY_HIGH;
    GVL_STATUS.G_Previous_Scenario := GVL_STATUS.G_Current_Scenario;

ELSIF GVL_STATUS.G_Diagnostics.Alarm_Event_Pulse THEN
    L_History_Write_Event := TRUE;
    L_History_Event.event_code := TO_WORD(GVL_STATUS.G_Diagnostics.Alarm_Event_Code);
    L_History_Event.event_value := GVL_STATUS.G_Diagnostics.Alarm_Event_Value;
    L_History_Event.unit := 10;
    L_History_Event.zone_id := 0;
    L_History_Event.priority := E_ALERT_PRIORITY.ALERT_PRIORITY_HIGH;

ELSIF GVL_STATUS.G_Diagnostics.Operator_Journal_Event_Seq <> L_Last_Operator_Journal_Seq THEN
    L_History_Write_Event := TRUE;
    L_History_Event.event_code := 1301;
    L_History_Event.event_value := TO_REAL(GVL_STATUS.G_Diagnostics.Operator_Journal_Event_Seq);
    L_History_Event.unit := 20;
    L_History_Event.zone_id := 0;
    L_History_Event.priority := E_ALERT_PRIORITY.ALERT_PRIORITY_HIGH;
    L_Last_Operator_Journal_Seq := GVL_STATUS.G_Diagnostics.Operator_Journal_Event_Seq;
END_IF;

IF L_History_Write_Event THEN
    IF (L_History_Event.event_code = L_Last_Event_Code)
       AND (ABS(L_History_Event.event_value - L_Last_Event_Value) < 0.001)
       AND (GVL_TIME_SERVICE.G_Now_MS - L_Last_Event_Time_MS < 5000) THEN
        L_History_Write_Event := FALSE;
    ELSE
        L_Last_Event_Code := L_History_Event.event_code;
        L_Last_Event_Value := L_History_Event.event_value;
        L_Last_Event_Time_MS := GVL_TIME_SERVICE.G_Now_MS;
    END_IF;
END_IF;

fbHistoryManager(
    VI_System_Time_MS := GVL_TIME_SERVICE.G_Now_MS,
    VI_Write_Event := L_History_Write_Event,
    VI_Event := L_History_Event
);
          
END_PROGRAM

PROGRAM PRG_Distributed_Domain

            // CANONICAL EXECUTION DOMAIN
// PRESERVES EXECUTION ORDER

PRG_Distributed_Peer_Ingestion();
PRG_Distributed_Epoch_Governor();
PRG_Distributed_Snapshot_Governor();
PRG_Distributed_Runtime_Supervisor();
PRG_Distributed_Commit_Governor();
          
END_PROGRAM

PROGRAM PRG_Behavior_Adapt_Profile

            // Centralized tuning profile controller.
// This block enforces consistent adaptive behavior settings.

CASE GVL_BEHAVIOR_ADAPT.G_Adapt_Profile OF

    ADAPT_PROFILE_STABLE:
        GVL_BEHAVIOR_ADAPT.G_Adapt_Learning_Rate := 0.03;
        GVL_BEHAVIOR_ADAPT.G_Confidence_Learning_Rate := 0.03;
        GVL_BEHAVIOR_ADAPT.G_Decay_Factor := 0.998;
        GVL_BEHAVIOR_ADAPT.G_Adapt_Update_Threshold := 7;

        GVL_BEHAVIOR_ADAPT.G_Behavior_Weight_Comfort := 1.0;
        GVL_BEHAVIOR_ADAPT.G_Behavior_Weight_Night := 1.0;
        GVL_BEHAVIOR_ADAPT.G_Behavior_Weight_Preheat := 1.0;
        GVL_BEHAVIOR_ADAPT.G_Behavior_Weight_VentBoost := 0.9;
        GVL_BEHAVIOR_ADAPT.G_Behavior_Weight_AccessSecure := 1.0;

    ADAPT_PROFILE_BALANCED:
        GVL_BEHAVIOR_ADAPT.G_Adapt_Learning_Rate := 0.05;
        GVL_BEHAVIOR_ADAPT.G_Confidence_Learning_Rate := 0.05;
        GVL_BEHAVIOR_ADAPT.G_Decay_Factor := 0.995;
        GVL_BEHAVIOR_ADAPT.G_Adapt_Update_Threshold := 5;

        GVL_BEHAVIOR_ADAPT.G_Behavior_Weight_Comfort := 1.0;
        GVL_BEHAVIOR_ADAPT.G_Behavior_Weight_Night := 1.0;
        GVL_BEHAVIOR_ADAPT.G_Behavior_Weight_Preheat := 1.0;
        GVL_BEHAVIOR_ADAPT.G_Behavior_Weight_VentBoost := 1.0;
        GVL_BEHAVIOR_ADAPT.G_Behavior_Weight_AccessSecure := 1.0;

    ADAPT_PROFILE_AGGRESSIVE:
        GVL_BEHAVIOR_ADAPT.G_Adapt_Learning_Rate := 0.08;
        GVL_BEHAVIOR_ADAPT.G_Confidence_Learning_Rate := 0.08;
        GVL_BEHAVIOR_ADAPT.G_Decay_Factor := 0.990;
        GVL_BEHAVIOR_ADAPT.G_Adapt_Update_Threshold := 3;

        GVL_BEHAVIOR_ADAPT.G_Behavior_Weight_Comfort := 1.0;
        GVL_BEHAVIOR_ADAPT.G_Behavior_Weight_Night := 1.0;
        GVL_BEHAVIOR_ADAPT.G_Behavior_Weight_Preheat := 1.0;
        GVL_BEHAVIOR_ADAPT.G_Behavior_Weight_VentBoost := 1.1;
        GVL_BEHAVIOR_ADAPT.G_Behavior_Weight_AccessSecure := 1.0;

ELSE
        // No fallback required
END_CASE;

// >>> BULK_SYNC_ANCHOR: PRG_Behavior_Adapt_Profile <<<
          
END_PROGRAM

PROGRAM PRG_Water_Output_Projection
  VAR
    fbWaterOutputProjector : FB_Water_Output_Projector;
    fbWaterOutputReconciliation : FB_Water_Output_Reconciliation;
    fbWaterValveFeedback : FB_Water_Valve_Feedback_Runtime;
    fbWaterPhysicalRuntime : FB_Water_Physical_Runtime;
    fbWaterRuntimeHardening : FB_Water_Runtime_Hardening;
    fbWaterRecoveryRuntime : FB_Water_Recovery_Runtime;
    fbPredictiveDiagnostics : FB_Predictive_Diagnostics_Runtime;
    fbForensicJournal : FB_Forensic_Journal_Runtime;
  END_VAR

            // Deterministic output projection runtime boundary.
//
// Runtime chain:
// output projection
//   -> reconciliation
//   -> valve feedback
//   -> physical convergence runtime
//   -> runtime hardening
//   -> recovery governance
//   -> predictive diagnostics
//   -> forensic journal
//
// No semantic/runtime authority.
// Existing global safety path preserved.

fbWaterOutputProjector(
    VI_Enable := TRUE,
    VI_System_Time_MS := GVL_STATUS.G_System_Time_MS
);

fbWaterOutputReconciliation(
    VI_Enable := TRUE,
    VI_System_Time_MS := GVL_STATUS.G_System_Time_MS
);

fbWaterValveFeedback(
    VI_Enable := TRUE,
    VI_System_Time_MS := GVL_STATUS.G_System_Time_MS
);

fbWaterPhysicalRuntime(
    VI_Enable := TRUE,
    VI_System_Time_MS := GVL_STATUS.G_System_Time_MS
);

fbWaterRuntimeHardening(
    VI_Enable := TRUE,
    VI_System_Time_MS := GVL_STATUS.G_System_Time_MS
);

fbWaterRecoveryRuntime(
    VI_Enable := TRUE,
    VI_System_Time_MS := GVL_STATUS.G_System_Time_MS
);

fbPredictiveDiagnostics(
    VI_Enable := TRUE,
    VI_System_Time_MS := GVL_STATUS.G_System_Time_MS
);

fbForensicJournal(
    VI_Enable := TRUE,
    VI_System_Time_MS := GVL_STATUS.G_System_Time_MS
);

// Runtime bridge integrated in PRG_Water.
// This PRG remains the deterministic projection boundary.
          
END_PROGRAM

PROGRAM PRG_Energy_Causality_Governor
  VAR
    L_Now_MS : UDINT;
    L_Energy_Valid : BOOL := TRUE;
    L_Error_Code : UDINT := 0;
    L_Error_Text : STRING(160) := '';
  END_VAR

            L_Now_MS := GVL_STATUS.G_System_Time_MS;
L_Energy_Valid := TRUE;
L_Error_Code := 0;
L_Error_Text := '';

// Fail-safe defaults.
GVL_ENERGY_CAUSALITY_FABRIC.Energy_Causality_Valid := FALSE;
GVL_ENERGY_CAUSALITY_FABRIC.Energy_Causality_Granted := FALSE;
GVL_ENERGY_CAUSALITY_FABRIC.Energy_Causality_Quarantine_Active := TRUE;

GVL_ENERGY_CAUSALITY_FABRIC.Hydraulic_Energy_State_Valid := FALSE;
GVL_ENERGY_CAUSALITY_FABRIC.Thermal_Energy_State_Valid := FALSE;
GVL_ENERGY_CAUSALITY_FABRIC.Electrical_Load_State_Valid := FALSE;
GVL_ENERGY_CAUSALITY_FABRIC.Motor_Energy_Envelope_Valid := FALSE;
GVL_ENERGY_CAUSALITY_FABRIC.Distributed_Load_Coherent := FALSE;

// Actuator semantic verification required.
IF NOT GVL_ACTUATOR_SEMANTIC_VERIFICATION.Actuator_Semantic_Verification_Granted THEN
    L_Energy_Valid := FALSE;
    L_Error_Code := 37000;
    L_Error_Text := 'Actuator semantic verification not granted';
END_IF;

// Energy divergence detectors.
IF GVL_ENERGY_CAUSALITY_FABRIC.DryRun_Energy_State_Detected THEN
    L_Energy_Valid := FALSE;
    L_Error_Code := 37001;
    L_Error_Text := 'Dry-run energy state detected';
END_IF;

IF GVL_ENERGY_CAUSALITY_FABRIC.Thermal_Extraction_Divergence_Detected THEN
    L_Energy_Valid := FALSE;
    L_Error_Code := 37002;
    L_Error_Text := 'Thermal extraction divergence detected';
END_IF;

IF GVL_ENERGY_CAUSALITY_FABRIC.Load_Synchronization_Spike_Detected THEN
    L_Energy_Valid := FALSE;
    L_Error_Code := 37003;
    L_Error_Text := 'Load synchronization spike detected';
END_IF;

IF GVL_ENERGY_CAUSALITY_FABRIC.Hydraulic_Energy_Starvation_Detected THEN
    L_Energy_Valid := FALSE;
    L_Error_Code := 37004;
    L_Error_Text := 'Hydraulic energy starvation detected';
END_IF;

IF GVL_ENERGY_CAUSALITY_FABRIC.Distributed_Transient_Overload_Detected THEN
    L_Energy_Valid := FALSE;
    L_Error_Code := 37005;
    L_Error_Text := 'Distributed transient overload detected';
END_IF;

IF GVL_ENERGY_CAUSALITY_FABRIC.Energy_Recovery_Instability_Detected THEN
    L_Energy_Valid := FALSE;
    L_Error_Code := 37006;
    L_Error_Text := 'Energy recovery instability detected';
END_IF;

// Stable energy envelope validation.
IF L_Energy_Valid
AND NOT GVL_ENERGY_CAUSALITY_FABRIC.Energy_Envelope_Stable THEN
    L_Energy_Valid := FALSE;
    L_Error_Code := 37010;
    L_Error_Text := 'Energy envelope unstable';
END_IF;

IF L_Energy_Valid
AND NOT GVL_ENERGY_CAUSALITY_FABRIC.Transient_Load_Stable THEN
    L_Energy_Valid := FALSE;
    L_Error_Code := 37011;
    L_Error_Text := 'Transient load stability invalid';
END_IF;

IF L_Energy_Valid
AND NOT GVL_ENERGY_CAUSALITY_FABRIC.Thermal_Accumulation_Stable THEN
    L_Energy_Valid := FALSE;
    L_Error_Code := 37012;
    L_Error_Text := 'Thermal accumulation unstable';
END_IF;

IF L_Energy_Valid
AND NOT GVL_ENERGY_CAUSALITY_FABRIC.Recovery_Energy_Coherent THEN
    L_Energy_Valid := FALSE;
    L_Error_Code := 37013;
    L_Error_Text := 'Recovery energy coherence invalid';
END_IF;

IF L_Energy_Valid THEN
    GVL_ENERGY_CAUSALITY_FABRIC.Energy_Causality_Valid := TRUE;
    GVL_ENERGY_CAUSALITY_FABRIC.Energy_Causality_Granted := TRUE;
    GVL_ENERGY_CAUSALITY_FABRIC.Energy_Causality_Quarantine_Active := FALSE;

    GVL_ENERGY_CAUSALITY_FABRIC.Hydraulic_Energy_State_Valid := TRUE;
    GVL_ENERGY_CAUSALITY_FABRIC.Thermal_Energy_State_Valid := TRUE;
    GVL_ENERGY_CAUSALITY_FABRIC.Electrical_Load_State_Valid := TRUE;
    GVL_ENERGY_CAUSALITY_FABRIC.Motor_Energy_Envelope_Valid := TRUE;
    GVL_ENERGY_CAUSALITY_FABRIC.Distributed_Load_Coherent := TRUE;

    GVL_ENERGY_CAUSALITY_FABRIC.Energy_Causality_Epoch :=
        GVL_ACTUATOR_SEMANTIC_VERIFICATION.Actuator_Verification_Epoch;

    GVL_ENERGY_CAUSALITY_FABRIC.Energy_Causality_Epoch_Coherent := TRUE;

    GVL_ENERGY_CAUSALITY_FABRIC.Energy_Causality_Last_Update_MS :=
        L_Now_MS;

    GVL_ENERGY_CAUSALITY_FABRIC.Energy_Causality_Lease_Expired := FALSE;

    GVL_ENERGY_CAUSALITY_FABRIC.Energy_Causality_Last_Error_Code := 0;
    GVL_ENERGY_CAUSALITY_FABRIC.Energy_Causality_Last_Error_Text := '';
ELSE
    GVL_ENERGY_CAUSALITY_FABRIC.Energy_Causality_Valid := FALSE;
    GVL_ENERGY_CAUSALITY_FABRIC.Energy_Causality_Granted := FALSE;
    GVL_ENERGY_CAUSALITY_FABRIC.Energy_Causality_Quarantine_Active := TRUE;

    GVL_ENERGY_CAUSALITY_FABRIC.Energy_Causality_Lease_Expired := TRUE;

    GVL_ENERGY_CAUSALITY_FABRIC.Energy_Causality_Last_Error_Code :=
        L_Error_Code;

    GVL_ENERGY_CAUSALITY_FABRIC.Energy_Causality_Last_Error_Text :=
        L_Error_Text;

    GVL_ENERGY_CAUSALITY_FABRIC.Energy_Causality_Invalidation_Count :=
        GVL_ENERGY_CAUSALITY_FABRIC.Energy_Causality_Invalidation_Count + 1;
END_IF;
          
END_PROGRAM

PROGRAM PRG_Modbus_Register_Scan
  VAR
    L_Register : UINT;
  END_VAR

            // ======================================================
// SAFE READ-ONLY MODBUS REGISTER SCAN
// ======================================================
// Safety rules:
//   - FC03/FC04 only.
//   - Never write registers.
//   - Manual enable only.
//   - Limited scan range.
// ======================================================

IF NOT GVL_MODBUS_SCAN.G_Scan_Enable THEN
    GVL_MODBUS_SCAN.G_Scan_Active := FALSE;
    GVL_MODBUS_SCAN.G_Scan_Done := FALSE;
    RETURN;
END_IF;

GVL_MODBUS_SCAN.G_Scan_Active := TRUE;
GVL_MODBUS_SCAN.G_Scan_Error := FALSE;

IF GVL_MODBUS_SCAN.G_Current_Register < GVL_MODBUS_SCAN.G_Start_Register THEN
    GVL_MODBUS_SCAN.G_Current_Register :=
        GVL_MODBUS_SCAN.G_Start_Register;
END_IF;

IF GVL_MODBUS_SCAN.G_Current_Register > GVL_MODBUS_SCAN.G_End_Register THEN
    GVL_MODBUS_SCAN.G_Scan_Active := FALSE;
    GVL_MODBUS_SCAN.G_Scan_Done := TRUE;
    RETURN;
END_IF;

L_Register := GVL_MODBUS_SCAN.G_Current_Register;

// ======================================================
// Issue read-only FC03 request
// ======================================================
GVL_MODBUS_MASTER.G_Request[16].Enable := TRUE;
GVL_MODBUS_MASTER.G_Request[16].Slave_ID := GVL_MODBUS_SCAN.G_Slave_ID;
GVL_MODBUS_MASTER.G_Request[16].Function_Code := MB_FC03_READ_HOLDING_REGISTERS;
GVL_MODBUS_MASTER.G_Request[16].Start_Register := L_Register;
GVL_MODBUS_MASTER.G_Request[16].Register_Count := 1;
GVL_MODBUS_MASTER.G_Request[16].Sequence :=
    GVL_MODBUS_MASTER.G_Request[16].Sequence + 1;
GVL_MODBUS_MASTER.G_Request[16].Timeout_MS := 250;

// ======================================================
// Process response
// ======================================================
IF GVL_MODBUS_MASTER.G_Response[16].Done THEN

    GVL_MODBUS_SCAN.G_Found_Register[L_Register] := TRUE;

    GVL_MODBUS_SCAN.G_Found_Value[L_Register] :=
        GVL_MODBUS_MASTER.G_Response[16].Read_Value[1];

    GVL_MODBUS_SCAN.G_Last_Scan_MS := GVL_STATUS.G_System_Time_MS;

    GVL_MODBUS_SCAN.G_Current_Register :=
        GVL_MODBUS_SCAN.G_Current_Register + 1;

ELSIF GVL_MODBUS_MASTER.G_Response[16].Error THEN

    GVL_MODBUS_SCAN.G_Found_Register[L_Register] := FALSE;

    GVL_MODBUS_SCAN.G_Current_Register :=
        GVL_MODBUS_SCAN.G_Current_Register + 1;

END_IF;
          
END_PROGRAM

PROGRAM PRG_Explainability
  VAR
    L_Mode : E_Safety_Mode;
    L_Recovery : E_Recovery_Phase;
    L_Command : STRING(120);
    L_Heating : STRING(255);
  END_VAR

            L_Mode := GVL_SAFETY_SHUTDOWN.G_Safety_Mode;
L_Recovery := GVL_SAFETY_RECOVERY.G_Recovery_Phase;

GVL_EXPLAINABILITY.G_Last_Safety_Mode := L_Mode;
GVL_EXPLAINABILITY.G_Last_Recovery_Phase := L_Recovery;
GVL_EXPLAINABILITY.G_Last_Update_MS := GVL_TIME_SERVICE.G_Now_MS;

// SAFETY LEVEL
CASE L_Mode OF
    FIRE: GVL_EXPLAINABILITY.G_Reason_Chain_Safety := 'FIRE';
    GAS: GVL_EXPLAINABILITY.G_Reason_Chain_Safety := 'GAS';
    WATER_LEAK: GVL_EXPLAINABILITY.G_Reason_Chain_Safety := 'WATER';
    GLOBAL_STOP: GVL_EXPLAINABILITY.G_Reason_Chain_Safety := 'GLOBAL_STOP';
    ELSE
        IF GVL_SAFETY_RECOVERY.G_Recovery_Active THEN
            GVL_EXPLAINABILITY.G_Reason_Chain_Safety := 'RECOVERY';
        ELSE
            GVL_EXPLAINABILITY.G_Reason_Chain_Safety := 'NORMAL';
        END_IF;
END_CASE;

// BEHAVIOR LEVEL
GVL_EXPLAINABILITY.G_Reason_Chain_Behavior := GVL_INTENT_BEHAVIOR.I_Reason_Text;

// COMMAND LEVEL
IF GVL_COMMAND_SHADOW.G_Heating_Block THEN
    L_Command := 'Heating Blocked';
ELSIF GVL_COMMAND_SHADOW.G_Vent_Stop THEN
    L_Command := 'Vent Stopped';
ELSIF GVL_COMMAND_SHADOW.G_Water_Block THEN
    L_Command := 'Water Blocked';
ELSE
    L_Command := 'Command OK';
END_IF;
GVL_EXPLAINABILITY.G_Reason_Chain_Command := L_Command;

// HEATING DOMAIN EXPLAINABILITY
IF GVL_STATE.G_Heating_RootCause <> E_Heating_RootCause.RC_NONE THEN
    L_Heating := GVL_STATE.G_Heating_Confidence_Reason_Text;
ELSIF GVL_STATE.G_Heating_Cascade_Degraded THEN
    L_Heating := 'Heating cascade degraded';
ELSE
    L_Heating := 'Heating OK';
END_IF;
GVL_EXPLAINABILITY.G_Heating_Why_Blocked := L_Heating;

// OUTPUT LEVEL
GVL_EXPLAINABILITY.G_Reason_Chain_Output := 'Outputs Applied';

// FULL CHAIN
GVL_EXPLAINABILITY.G_Reason_Chain_Full := CONCAT(
    CONCAT(
        CONCAT(
            GVL_EXPLAINABILITY.G_Reason_Chain_Safety,
            ' -> '
        ),
        CONCAT(
            GVL_EXPLAINABILITY.G_Reason_Chain_Behavior,
            ' -> '
        )
    ),
    CONCAT(
        CONCAT(
            GVL_EXPLAINABILITY.G_Reason_Chain_Command,
            ' -> '
        ),
        CONCAT(
            L_Heating,
            ' -> Outputs Applied'
        )
    )
);

// KEEP OLD FIELDS
GVL_EXPLAINABILITY.G_Behavior_Why_Active := GVL_INTENT_BEHAVIOR.I_Reason_Text;
          
END_PROGRAM

PROGRAM PRG_Resource_Starvation_Boundary_Governor

            IF GVL_EXECUTION_PROGRESS_CAUSALITY_FABRIC.Execution_Progress_Causality_Granted
AND NOT GVL_RESOURCE_STARVATION_BOUNDARY_FABRIC.Resource_Starvation_Detected
AND NOT GVL_RESOURCE_STARVATION_BOUNDARY_FABRIC.Scheduler_Starvation_Detected
AND NOT GVL_RESOURCE_STARVATION_BOUNDARY_FABRIC.Distributed_Allocation_Deadlock_Detected THEN

    GVL_RESOURCE_STARVATION_BOUNDARY_FABRIC.Resource_Starvation_Boundary_Valid := TRUE;
    GVL_RESOURCE_STARVATION_BOUNDARY_FABRIC.Resource_Starvation_Boundary_Granted := TRUE;
    GVL_RESOURCE_STARVATION_BOUNDARY_FABRIC.Resource_Starvation_Bounded := TRUE;
    GVL_RESOURCE_STARVATION_BOUNDARY_FABRIC.Fair_Execution_Scheduling_Valid := TRUE;
END_IF;
          
END_PROGRAM

PROGRAM PRG_Semantic_Commit_Governor
  VAR
    L_Now_MS : UDINT;
    L_Delta_MS : UDINT;
    L_Commit_Valid : BOOL := TRUE;
    L_Error_Code : UDINT := 0;
    L_Error_Text : STRING(160) := '';
  END_VAR

            L_Now_MS := GVL_STATUS.G_System_Time_MS;
L_Commit_Valid := TRUE;
L_Error_Code := 0;
L_Error_Text := '';

// ======================================================
// SEMANTIC PUBLICATION COMMIT GOVERNOR
// ======================================================
// Governs semantic publication checkpoint coherence.
// Downstream/publication continuity only.
// Does not invalidate runtime barrier, PLC fencing,
// immutable snapshots, distributed commit or IO authority.
// ======================================================

GVL_SEMANTIC_COMMIT.Semantic_Checkpoint_Mismatch := FALSE;
GVL_SEMANTIC_COMMIT.Semantic_Commit_Mismatch := FALSE;
GVL_SEMANTIC_COMMIT.Semantic_Rollback_Detected := FALSE;
GVL_SEMANTIC_COMMIT.Semantic_Replay_Fenced := FALSE;
GVL_SEMANTIC_COMMIT.Semantic_Checkpoint_Missing := FALSE;
GVL_SEMANTIC_COMMIT.Semantic_Commit_Lease_Expired := FALSE;

// ------------------------------------------------------
// Semantic checkpoint epoch progression.
// ------------------------------------------------------

GVL_SEMANTIC_COMMIT.Local_Semantic_Checkpoint_Epoch :=
    GVL_SEMANTIC_COMMIT.Local_Semantic_Checkpoint_Epoch + 1;

GVL_SEMANTIC_COMMIT.Local_Semantic_Commit_Epoch :=
    GVL_SEMANTIC_COMMIT.Local_Semantic_Commit_Epoch + 1;

// ------------------------------------------------------
// Rollback/replay fencing foundation.
// ------------------------------------------------------

IF GVL_SEMANTIC_COMMIT.Peer_Semantic_Checkpoint_Epoch
< GVL_SEMANTIC_COMMIT.Local_Semantic_Checkpoint_Epoch THEN
    GVL_SEMANTIC_COMMIT.Semantic_Rollback_Detected := TRUE;
    GVL_SEMANTIC_COMMIT.Semantic_Replay_Fenced := TRUE;

    L_Commit_Valid := FALSE;
    L_Error_Code := 18000;
    L_Error_Text := 'Semantic rollback detected';
END_IF;

// ------------------------------------------------------
// Checkpoint acknowledgement foundation.
// ------------------------------------------------------

IF L_Commit_Valid THEN
    IF NOT GVL_SEMANTIC_COMMIT.Semantic_Checkpoint_Ack_Valid THEN
        GVL_SEMANTIC_COMMIT.Semantic_Checkpoint_Missing := TRUE;

        L_Commit_Valid := FALSE;
        L_Error_Code := 18001;
        L_Error_Text := 'Semantic checkpoint acknowledgement missing';
    END_IF;
END_IF;

// ------------------------------------------------------
// Semantic checkpoint mismatch foundation.
// ------------------------------------------------------

IF L_Commit_Valid THEN
    IF GVL_SEMANTIC_COMMIT.Peer_Semantic_Commit_Epoch
    <> GVL_SEMANTIC_COMMIT.Local_Semantic_Commit_Epoch THEN
        GVL_SEMANTIC_COMMIT.Semantic_Commit_Mismatch := TRUE;

        L_Commit_Valid := FALSE;
        L_Error_Code := 18002;
        L_Error_Text := 'Semantic commit mismatch detected';
    END_IF;
END_IF;

// ------------------------------------------------------
// Semantic commit lease freshness.
// ------------------------------------------------------

L_Delta_MS :=
    L_Now_MS - GVL_SEMANTIC_COMMIT.Semantic_Commit_Last_Refresh_MS;

IF L_Commit_Valid
AND GVL_SEMANTIC_COMMIT.Semantic_Commit_Lease_Active THEN
    IF L_Delta_MS > GVL_SEMANTIC_COMMIT.Semantic_Commit_Timeout_MS THEN
        GVL_SEMANTIC_COMMIT.Semantic_Commit_Lease_Expired := TRUE;

        L_Commit_Valid := FALSE;
        L_Error_Code := 18003;
        L_Error_Text := 'Semantic commit lease expired';
    END_IF;
END_IF;

// ------------------------------------------------------
// Publish semantic commit coherence foundation.
// ------------------------------------------------------

IF L_Commit_Valid THEN
    GVL_SEMANTIC_COMMIT.Semantic_Commit_Epoch :=
        GVL_SEMANTIC_COMMIT.Semantic_Commit_Epoch + 1;

    GVL_SEMANTIC_COMMIT.Semantic_Checkpoint_Epoch :=
        GVL_SEMANTIC_COMMIT.Semantic_Checkpoint_Epoch + 1;

    GVL_SEMANTIC_COMMIT.Semantic_Publication_Commit_Epoch :=
        GVL_SEMANTIC_COMMIT.Semantic_Publication_Commit_Epoch + 1;

    GVL_SEMANTIC_COMMIT.Semantic_Commit_Valid := TRUE;
    GVL_SEMANTIC_COMMIT.Semantic_Commit_Lease_Active := TRUE;
    GVL_SEMANTIC_COMMIT.Semantic_Commit_Lease_Expired := FALSE;

    GVL_SEMANTIC_COMMIT.Semantic_Commit_Quarantine_Active := FALSE;
    GVL_SEMANTIC_COMMIT.Semantic_Commit_Forced_Safe_Mode := FALSE;

    GVL_SEMANTIC_COMMIT.Semantic_Commit_Last_Refresh_MS := L_Now_MS;

    GVL_SEMANTIC_COMMIT.Semantic_Commit_Last_Error_Code := 0;
    GVL_SEMANTIC_COMMIT.Semantic_Commit_Last_Error_Text := '';
ELSE
    GVL_SEMANTIC_COMMIT.Semantic_Commit_Valid := FALSE;
    GVL_SEMANTIC_COMMIT.Semantic_Commit_Quarantine_Active := TRUE;
    GVL_SEMANTIC_COMMIT.Semantic_Commit_Forced_Safe_Mode := TRUE;

    GVL_SEMANTIC_COMMIT.Semantic_Commit_Last_Error_Code := L_Error_Code;
    GVL_SEMANTIC_COMMIT.Semantic_Commit_Last_Error_Text := L_Error_Text;

    GVL_SEMANTIC_COMMIT.Semantic_Commit_Invalidation_Count :=
        GVL_SEMANTIC_COMMIT.Semantic_Commit_Invalidation_Count + 1;
END_IF;
          
END_PROGRAM

PROGRAM PRG_Physical_Authority_Epoch_Governor
  VAR
    L_Now_MS : UDINT;
    L_Epoch_Valid : BOOL := TRUE;
    L_Error_Code : UDINT := 0;
    L_Error_Text : STRING(160) := '';
    L_Global_Epoch : UDINT;
  END_VAR

            L_Now_MS := GVL_STATUS.G_System_Time_MS;
L_Epoch_Valid := TRUE;
L_Error_Code := 0;
L_Error_Text := '';

// Fail-safe defaults.
GVL_PHYSICAL_AUTHORITY_EPOCH.Physical_Authority_Epoch_Valid := FALSE;
GVL_PHYSICAL_AUTHORITY_EPOCH.Snapshot_Epoch_Coherent := FALSE;
GVL_PHYSICAL_AUTHORITY_EPOCH.Consensus_Epoch_Coherent := FALSE;
GVL_PHYSICAL_AUTHORITY_EPOCH.Causality_Epoch_Coherent := FALSE;
GVL_PHYSICAL_AUTHORITY_EPOCH.PreOutput_Epoch_Coherent := FALSE;

L_Global_Epoch := GVL_PHYSICAL_SNAPSHOT.Physical_Snapshot_Epoch;

// Snapshot epoch is the authoritative physical world epoch.
IF GVL_PHYSICAL_SNAPSHOT.Physical_Snapshot_Epoch = 0 THEN
    L_Epoch_Valid := FALSE;
    L_Error_Code := 24000;
    L_Error_Text := 'Physical snapshot epoch invalid';
END_IF;

// Consensus must validate the same immutable world.
IF L_Epoch_Valid
AND (GVL_SENSOR_CONSENSUS.Sensor_Consensus_Epoch <> L_Global_Epoch) THEN
    GVL_PHYSICAL_AUTHORITY_EPOCH.Cross_Cycle_Epoch_Skew_Detected := TRUE;

    L_Epoch_Valid := FALSE;
    L_Error_Code := 24001;
    L_Error_Text := 'Sensor consensus epoch skew detected';
END_IF;

// Telemetry causality must validate the same immutable world.
IF L_Epoch_Valid
AND (GVL_TELEMETRY.Telemetry_Epoch <> L_Global_Epoch) THEN
    GVL_PHYSICAL_AUTHORITY_EPOCH.Cross_Cycle_Epoch_Skew_Detected := TRUE;

    L_Epoch_Valid := FALSE;
    L_Error_Code := 24002;
    L_Error_Text := 'Telemetry epoch skew detected';
END_IF;

// Output publication epoch must remain coherent.
IF L_Epoch_Valid
AND (GVL_OUTPUT_EPOCH.Output_Publication_Epoch <> L_Global_Epoch) THEN
    GVL_PHYSICAL_AUTHORITY_EPOCH.Partial_Epoch_Advancement_Detected := TRUE;

    L_Epoch_Valid := FALSE;
    L_Error_Code := 24003;
    L_Error_Text := 'Output publication epoch skew detected';
END_IF;

IF L_Epoch_Valid
AND GVL_PHYSICAL_AUTHORITY_EPOCH.Physical_Epoch_Replay_Suspected THEN
    L_Epoch_Valid := FALSE;
    L_Error_Code := 24004;
    L_Error_Text := 'Physical authority epoch replay suspected';
END_IF;

IF L_Epoch_Valid
AND GVL_PHYSICAL_AUTHORITY_EPOCH.Physical_Epoch_Drift_Detected THEN
    L_Epoch_Valid := FALSE;
    L_Error_Code := 24005;
    L_Error_Text := 'Physical authority epoch drift detected';
END_IF;

IF L_Epoch_Valid THEN
    GVL_PHYSICAL_AUTHORITY_EPOCH.Physical_Authority_Epoch := L_Global_Epoch;
    GVL_PHYSICAL_AUTHORITY_EPOCH.Physical_Authority_Epoch_Valid := TRUE;

    GVL_PHYSICAL_AUTHORITY_EPOCH.Snapshot_Epoch_Coherent := TRUE;
    GVL_PHYSICAL_AUTHORITY_EPOCH.Consensus_Epoch_Coherent := TRUE;
    GVL_PHYSICAL_AUTHORITY_EPOCH.Causality_Epoch_Coherent := TRUE;
    GVL_PHYSICAL_AUTHORITY_EPOCH.PreOutput_Epoch_Coherent := TRUE;

    GVL_PHYSICAL_AUTHORITY_EPOCH.Physical_Authority_Lease_Expired := FALSE;
    GVL_PHYSICAL_AUTHORITY_EPOCH.Physical_Authority_Quarantine_Active := FALSE;

    GVL_PHYSICAL_AUTHORITY_EPOCH.Physical_Authority_Last_Update_MS := L_Now_MS;

    GVL_PHYSICAL_AUTHORITY_EPOCH.Physical_Authority_Last_Error_Code := 0;
    GVL_PHYSICAL_AUTHORITY_EPOCH.Physical_Authority_Last_Error_Text := '';
ELSE
    GVL_PHYSICAL_AUTHORITY_EPOCH.Physical_Authority_Epoch_Valid := FALSE;

    GVL_PHYSICAL_AUTHORITY_EPOCH.Physical_Authority_Lease_Expired := TRUE;
    GVL_PHYSICAL_AUTHORITY_EPOCH.Physical_Authority_Quarantine_Active := TRUE;

    GVL_PHYSICAL_AUTHORITY_EPOCH.Physical_Authority_Last_Error_Code := L_Error_Code;
    GVL_PHYSICAL_AUTHORITY_EPOCH.Physical_Authority_Last_Error_Text := L_Error_Text;

    GVL_PHYSICAL_AUTHORITY_EPOCH.Physical_Authority_Invalidation_Count :=
        GVL_PHYSICAL_AUTHORITY_EPOCH.Physical_Authority_Invalidation_Count + 1;
END_IF;
          
END_PROGRAM

PROGRAM PRG_Observability_Truth_Governor
  VAR
    L_Now_MS : UDINT;
    L_Observability_Valid : BOOL := TRUE;
    L_Error_Code : UDINT := 0;
    L_Error_Text : STRING(160) := '';
  END_VAR

            L_Now_MS := GVL_STATUS.G_System_Time_MS;
L_Observability_Valid := TRUE;
L_Error_Code := 0;
L_Error_Text := '';

// Fail-safe defaults.
GVL_OBSERVABILITY_TRUTH.Observability_Truth_Valid := FALSE;
GVL_OBSERVABILITY_TRUTH.Observability_Truth_Granted := FALSE;
GVL_OBSERVABILITY_TRUTH.Observability_Truth_Quarantine_Active := TRUE;

GVL_OBSERVABILITY_TRUTH.HMI_Authority_Coherent := FALSE;
GVL_OBSERVABILITY_TRUTH.Alarm_Authority_Coherent := FALSE;
GVL_OBSERVABILITY_TRUTH.Trend_Authority_Coherent := FALSE;
GVL_OBSERVABILITY_TRUTH.Diagnostics_Authority_Coherent := FALSE;
GVL_OBSERVABILITY_TRUTH.History_Authority_Coherent := FALSE;

// Semantic continuity authority required.
IF NOT GVL_SEMANTIC_CONTINUITY.Semantic_Continuity_Granted THEN
    L_Observability_Valid := FALSE;
    L_Error_Code := 32000;
    L_Error_Text := 'Semantic continuity authority not granted';
END_IF;

// Observability split-brain detectors.
IF GVL_OBSERVABILITY_TRUTH.Stale_HMI_Epoch_Detected THEN
    L_Observability_Valid := FALSE;
    L_Error_Code := 32001;
    L_Error_Text := 'Stale HMI epoch detected';
END_IF;

IF GVL_OBSERVABILITY_TRUTH.Alarm_Publication_Lag_Detected THEN
    L_Observability_Valid := FALSE;
    L_Error_Code := 32002;
    L_Error_Text := 'Alarm publication lag detected';
END_IF;

IF GVL_OBSERVABILITY_TRUTH.Trend_Causality_Skew_Detected THEN
    L_Observability_Valid := FALSE;
    L_Error_Code := 32003;
    L_Error_Text := 'Trend causality skew detected';
END_IF;

IF GVL_OBSERVABILITY_TRUTH.Diagnostic_Truth_Race_Detected THEN
    L_Observability_Valid := FALSE;
    L_Error_Code := 32004;
    L_Error_Text := 'Diagnostic truth race detected';
END_IF;

IF GVL_OBSERVABILITY_TRUTH.Operator_Visibility_Fragmentation_Detected THEN
    L_Observability_Valid := FALSE;
    L_Error_Code := 32005;
    L_Error_Text := 'Operator visibility fragmentation detected';
END_IF;

IF GVL_OBSERVABILITY_TRUTH.Authority_UI_Divergence_Detected THEN
    L_Observability_Valid := FALSE;
    L_Error_Code := 32006;
    L_Error_Text := 'Authority/UI divergence detected';
END_IF;

// Projection causality validation.
IF L_Observability_Valid
AND NOT GVL_OBSERVABILITY_TRUTH.HMI_Epoch_Coherent THEN
    L_Observability_Valid := FALSE;
    L_Error_Code := 32010;
    L_Error_Text := 'HMI epoch coherence invalid';
END_IF;

IF L_Observability_Valid
AND NOT GVL_OBSERVABILITY_TRUTH.Alarm_Publication_Coherent THEN
    L_Observability_Valid := FALSE;
    L_Error_Code := 32011;
    L_Error_Text := 'Alarm publication coherence invalid';
END_IF;

IF L_Observability_Valid
AND NOT GVL_OBSERVABILITY_TRUTH.Trend_Causality_Coherent THEN
    L_Observability_Valid := FALSE;
    L_Error_Code := 32012;
    L_Error_Text := 'Trend causality coherence invalid';
END_IF;

IF L_Observability_Valid
AND NOT GVL_OBSERVABILITY_TRUTH.Diagnostics_Causality_Coherent THEN
    L_Observability_Valid := FALSE;
    L_Error_Code := 32013;
    L_Error_Text := 'Diagnostics causality coherence invalid';
END_IF;

IF L_Observability_Valid
AND NOT GVL_OBSERVABILITY_TRUTH.Operator_Visibility_Consistent THEN
    L_Observability_Valid := FALSE;
    L_Error_Code := 32014;
    L_Error_Text := 'Operator visibility consistency invalid';
END_IF;

IF L_Observability_Valid THEN
    GVL_OBSERVABILITY_TRUTH.Observability_Truth_Valid := TRUE;
    GVL_OBSERVABILITY_TRUTH.Observability_Truth_Granted := TRUE;
    GVL_OBSERVABILITY_TRUTH.Observability_Truth_Quarantine_Active := FALSE;

    GVL_OBSERVABILITY_TRUTH.HMI_Authority_Coherent := TRUE;
    GVL_OBSERVABILITY_TRUTH.Alarm_Authority_Coherent := TRUE;
    GVL_OBSERVABILITY_TRUTH.Trend_Authority_Coherent := TRUE;
    GVL_OBSERVABILITY_TRUTH.Diagnostics_Authority_Coherent := TRUE;
    GVL_OBSERVABILITY_TRUTH.History_Authority_Coherent := TRUE;

    GVL_OBSERVABILITY_TRUTH.Observability_Truth_Epoch :=
        GVL_SEMANTIC_CONTINUITY.Semantic_Continuity_Epoch;

    GVL_OBSERVABILITY_TRUTH.Observability_Truth_Epoch_Coherent := TRUE;

    GVL_OBSERVABILITY_TRUTH.Observability_Last_Update_MS := L_Now_MS;
    GVL_OBSERVABILITY_TRUTH.Observability_Lease_Expired := FALSE;

    GVL_OBSERVABILITY_TRUTH.Observability_Last_Error_Code := 0;
    GVL_OBSERVABILITY_TRUTH.Observability_Last_Error_Text := '';
ELSE
    GVL_OBSERVABILITY_TRUTH.Observability_Truth_Valid := FALSE;
    GVL_OBSERVABILITY_TRUTH.Observability_Truth_Granted := FALSE;
    GVL_OBSERVABILITY_TRUTH.Observability_Truth_Quarantine_Active := TRUE;

    GVL_OBSERVABILITY_TRUTH.Observability_Lease_Expired := TRUE;

    GVL_OBSERVABILITY_TRUTH.Observability_Last_Error_Code :=
        L_Error_Code;

    GVL_OBSERVABILITY_TRUTH.Observability_Last_Error_Text :=
        L_Error_Text;

    GVL_OBSERVABILITY_TRUTH.Observability_Invalidation_Count :=
        GVL_OBSERVABILITY_TRUTH.Observability_Invalidation_Count + 1;
END_IF;
          
END_PROGRAM

PROGRAM PRG_Authority_Revocation_Governor
  VAR
    L_Now_MS : UDINT;
    L_Revocation_Required : BOOL := FALSE;
  END_VAR

            L_Now_MS := GVL_STATUS.G_System_Time_MS;

// Fail-safe defaults.
GVL_AUTHORITY_REVOCATION.Authority_Revocation_Active := FALSE;
GVL_AUTHORITY_REVOCATION.Authority_Revocation_Propagated := FALSE;
GVL_AUTHORITY_REVOCATION.Authority_Fail_Closed_Valid := FALSE;
GVL_AUTHORITY_REVOCATION.Revocation_Order_Valid := FALSE;

// Detect upstream authority invalidation.
GVL_AUTHORITY_REVOCATION.Snapshot_Authority_Revoked :=
    NOT GVL_PHYSICAL_SNAPSHOT.Physical_Snapshot_Valid;

GVL_AUTHORITY_REVOCATION.Sensor_Consensus_Authority_Revoked :=
    NOT GVL_SENSOR_CONSENSUS.Sensor_Consensus_Valid;

GVL_AUTHORITY_REVOCATION.Telemetry_Causality_Authority_Revoked :=
    NOT GVL_TELEMETRY.Command_Telemetry_Causality_Valid;

GVL_AUTHORITY_REVOCATION.Physical_Authority_Epoch_Revoked :=
    NOT GVL_PHYSICAL_AUTHORITY_EPOCH.Physical_Authority_Epoch_Valid;

GVL_AUTHORITY_REVOCATION.Authority_Lineage_Revoked :=
    NOT GVL_AUTHORITY_LINEAGE.Authority_Lineage_Valid;

L_Revocation_Required :=
    GVL_AUTHORITY_REVOCATION.Snapshot_Authority_Revoked
    OR GVL_AUTHORITY_REVOCATION.Sensor_Consensus_Authority_Revoked
    OR GVL_AUTHORITY_REVOCATION.Telemetry_Causality_Authority_Revoked
    OR GVL_AUTHORITY_REVOCATION.Physical_Authority_Epoch_Revoked
    OR GVL_AUTHORITY_REVOCATION.Authority_Lineage_Revoked;

IF L_Revocation_Required THEN
    GVL_AUTHORITY_REVOCATION.Authority_Revocation_Active := TRUE;
    GVL_AUTHORITY_REVOCATION.Quarantine_Fabric_Active := TRUE;

    GVL_AUTHORITY_REVOCATION.PreOutput_Authority_Revoked := TRUE;
    GVL_AUTHORITY_REVOCATION.Physical_IO_Release_Denied := TRUE;

    GVL_AUTHORITY_REVOCATION.Authority_Revocation_Propagated := TRUE;
    GVL_AUTHORITY_REVOCATION.Authority_Fail_Closed_Valid := TRUE;
    GVL_AUTHORITY_REVOCATION.Revocation_Order_Valid := TRUE;

    GVL_AUTHORITY_REVOCATION.Revocation_Epoch :=
        GVL_PHYSICAL_AUTHORITY_EPOCH.Physical_Authority_Epoch;

    GVL_AUTHORITY_REVOCATION.Revocation_Last_Update_MS := L_Now_MS;
ELSE
    GVL_AUTHORITY_REVOCATION.Authority_Revocation_Active := FALSE;
    GVL_AUTHORITY_REVOCATION.Quarantine_Fabric_Active := FALSE;

    GVL_AUTHORITY_REVOCATION.PreOutput_Authority_Revoked := FALSE;
    GVL_AUTHORITY_REVOCATION.Physical_IO_Release_Denied := FALSE;

    GVL_AUTHORITY_REVOCATION.Authority_Revocation_Propagated := FALSE;
    GVL_AUTHORITY_REVOCATION.Authority_Fail_Closed_Valid := TRUE;
    GVL_AUTHORITY_REVOCATION.Revocation_Order_Valid := TRUE;
END_IF;
          
END_PROGRAM

PROGRAM PRG_Runtime_Barrier
  VAR
    L_Now_MS : UDINT;
    L_Runtime_OK : BOOL := TRUE;
    L_Error_Code : UDINT := 0;
    L_Error_Text : STRING(160) := '';
    L_Finalized_Continuity_Healthy : BOOL;
  END_VAR

            L_Now_MS := GVL_STATUS.G_System_Time_MS;
L_Runtime_OK := TRUE;
L_Error_Code := 0;
L_Error_Text := '';

// ======================================================
// AUTHORITATIVE RUNTIME BARRIER
// ======================================================
// Creates authoritative runtime publication semantics.
// Rejects impossible runtime states before physical publication.
//
// Runtime authority remains:
// - monotonic-time authoritative;
// - PLC fencing authoritative;
// - transport freshness authoritative.
//
// Finalized distributed commit continuity is allowed
// as upstream authority evidence.
//
// Semantic continuity intentionally remains downstream
// to avoid primordial semantic/runtime recursion.
// ======================================================

GVL_RUNTIME_EPOCH.Runtime_Cycle_Start_MS := L_Now_MS;
GVL_RUNTIME_EPOCH.Runtime_Snapshot_Published := FALSE;
GVL_RUNTIME_EPOCH.Runtime_Impossible_State_Detected := FALSE;
GVL_RUNTIME_EPOCH.Runtime_IO_Publication_Allowed := FALSE;

IF NOT GVL_TIME_MONOTONIC.Monotonic_Time_Initialized THEN
    L_Runtime_OK := FALSE;
    L_Error_Code := 4900;
    L_Error_Text := 'Monotonic time not initialized';
END_IF;

IF L_Runtime_OK AND (NOT GVL_TIME_MONOTONIC.Monotonic_Time_Valid) THEN
    L_Runtime_OK := FALSE;
    L_Error_Code := 4901;
    L_Error_Text := 'Monotonic time invalid';
END_IF;

IF L_Runtime_OK AND GVL_TIME_MONOTONIC.Startup_Quarantine_Active THEN
    L_Runtime_OK := FALSE;
    L_Error_Code := 4902;
    L_Error_Text := 'Startup quarantine active';
END_IF;

IF L_Runtime_OK AND GVL_TIME_MONOTONIC.Time_Rollback_Detected THEN
    L_Runtime_OK := FALSE;
    L_Error_Code := 4903;
    L_Error_Text := 'Monotonic rollback detected';
END_IF;

IF L_Runtime_OK AND GVL_TIME_MONOTONIC.Retained_Time_Invalid THEN
    L_Runtime_OK := FALSE;
    L_Error_Code := 4904;
    L_Error_Text := 'Retained monotonic time invalid';
END_IF;

